// TwinCAT 3 PLC project PulsedPowerSlim_PLC
// ProgramVersion: 3.1.4023.0
// libraries:
//   Tc2_DataExchange, * (Beckhoff Automation GmbH)
//   Tc2_Math, * (Beckhoff Automation GmbH)
//   Tc2_Standard, * (Beckhoff Automation GmbH)
//   Tc2_System, * (Beckhoff Automation GmbH)
//   Tc3_EventLogger, * (Beckhoff Automation GmbH)
//   Tc3_Module, * (Beckhoff Automation GmbH)
// project tree:
//   DUTs/ E_PulseState.TcDUT, ST_Alarm_Base.TcDUT (not stored), ST_RelayFaults_Form.TcDUT, ST_Section_Base.TcDUT, ST_Charger_Base.TcDUT, ST_FieldDevices_Base.TcDUT, ST_InstrumentReading.TcDUT, ST_RelayFaults_Base.TcDUT, ST_FieldDevices_Form.TcDUT, ST_Trip_Base.TcDUT, ST_VoltageFeedback.TcDUT (not stored)
//   GVLs/ Alarms_DB.TcGVL, GVL.TcGVL, Input.TcGVL, LCP.TcGVL (not stored), MCP_IO.TcGVL, Output.TcGVL, Permissives_DB.TcGVL, Trips_DB.TcGVL
//   / PlcTask.TcTTO
//   POUs/ Alarms.TcPOU, Alarms_FB.TcPOU (not stored), Alias.TcPOU, Heartbeat.TcPOU (not stored), MAIN.TcPOU, Permissives.TcPOU, Sequence.TcPOU, Trips.TcPOU
// real-time tasks:
//   TASK PlcTask: cycle T#10ms, priority 20, ADS port 350

CONFIGURATION PulsedPowerSlim_PLC
    RESOURCE PLC ON TwinCAT3
        TASK PlcTask(INTERVAL := T#10ms, PRIORITY := 20);
        PROGRAM MAIN WITH PlcTask : MAIN;
    END_RESOURCE
END_CONFIGURATION

// ---- DUTs/E_PulseState.TcDUT
{attribute 'qualified_only'}
{attribute 'strict'}
TYPE E_PulseState :
(
	SAFE			:= 0, //IDLE
	CHARGING		:= 1, //Charge
	CHARGECOMPLETE	:= 2, //EOC
	//DISCONNECTING	:= 3, //Disconnect
	DUMPING			:= 4, 
	//ABORT			:= 5,
	TRIPPED			:= 6	
);
END_TYPE

// ---- DUTs/ST_RelayFaults_Form.TcDUT
TYPE ST_RelayFaults_Form EXTENDS ST_RelayFaults_Base :
STRUCT
	PreFormChrgRlyFailed				: BOOL;
	PreFormChrgRlyFaultDelay_TON		: TON;
	FormTrigChrgRlyFailed				: BOOL;
	FormTrigChrgRlyFaultDelay_TON		: TON;
	PreFormTrigChrgRlyFailed			: BOOL;
	PreFormTrigChrgRlyFaultDelay_TON	: TON;
	PreFormDumpRlyFailed				: BOOL;
	PreFormDumpRlyFaultDelay_TON		: TON;
	FormTrigDumpRly1Failed				: BOOL;
	FormTrigDumpRlyFaultDelay_TON		: TON;
	PreFormTrigDumpRly1Failed			: BOOL;
	PreFormTrigDumpRlyFaultDelay_TON	: TON;
END_STRUCT
END_TYPE

// ---- DUTs/ST_Section_Base.TcDUT
//Base coil type with all the Common functionality
TYPE ST_Section_Base :
STRUCT
	
	Peak : ST_FieldDevices_Base;
	Sust : ST_FieldDevices_Base;
	Form : ST_FieldDevices_Form;
	
	FormTriggerCapVoltage_raw				: INT;
	PSU1_DCOK								: BOOL := FALSE;
	//Local_EstopPB_Pressed					: BOOL;  //NC
	SystemReadyToCharge						: BOOL := FALSE;
	LossPneumaticPressure					: BOOL;
	
	//*********************************************************************************
	(*ChargeVoltageFeedback					: REAL;
	ChargeVoltageFeedback_raw				: INT;
	ChargerVoltageFeedback_norm				: REAL;
	
	CurrentFeedback							: REAL;
	CurrentFeedback_raw						: INT;
	CurrentFeedback_norm					: REAL;
	
	chargerSetpoint							: INT;  //0-100% analog PWM 24V output -> (0 - 10V)
	chargerSetpoint_norm					: REAL;
	chargerSetpoint_raw						: REAL;
	currentSetpoint							: INT;  //0-100% analog PWM 24V output -> (0.5 - 4.5V)
	currentSetpoint_norm					: REAL;
	currentSetpoint_raw						: REAL;
	//currentSetpointFromMaster: REAL;

	
	DumpRelay1_closed						: BOOL;
	DumpRelay2_closed						: BOOL;
	ChargeRelay_closed						: BOOL := FALSE;
	ChargerIsEnabled						: BOOL := FALSE; //feedback from charger
	FlybackD1_Alive							: BOOL := FALSE;
	FlybackD2_Alive							: BOOL := FALSE;
	
	DumpResistorTemperatureHigh				: BOOL; 
	GroundLoopCurrentDetected				: BOOL;
	CoilTemperatureHigh						: BOOL := FALSE;
	AC_Interlock_RlyClose					: BOOL;
	
	
	OpenDumpRelays							: BOOL := FALSE;
	closeChargeRelay						: BOOL := FALSE;
	enableOutputToCharger					: BOOL := FALSE;  //output going to charger
	CloseACInterlockRly						: BOOL := FALSE;
	SystemFaulted							: BOOL := FALSE;
	SystemCharging							: BOOL := FALSE;
	
	
	CoilEnabled								: BOOL := TRUE;
	
	NumOfCap								: INT := 4;
	
	//CoilSafetyOK							: BOOL;
	ChargerWarning							: BOOL;  //comes from UltraCaps CANBUS message
	CapVoltage								: INT;   //Comes from UlgraCaps CANBUS message
	
	ChargerVoltageFault_TON : TON;
	ChargerVoltageFault_ET : TIME;
	CurrentSensorFault_TON : TON;
	CurrentSensorFault_ET : TIME;
	BfieldSensorFault_TON : TON;
	BfieldSensorFault_ET : TIME;
	
	CAN_id: INT;
	CAN_AdsAddr: AMSADDR;
	CAN_netID: AMSNETID;
	CAN_port: WORD;
	CAN_error: USINT;
	CAN_State: UINT;
	CAN_RxErrorCounter: USINT;	
	CAN_TxErrorCounter: USINT;	
	CAN_DiagFlag: BOOL;
	
	UltacCap_CAN_error: USINT;
	UltraCap_CAN_State: UINT;
	UltraCap_CAN_RxErrorCounter: USINT;	
	UltraCap_CAN_TxErrorCounter: USINT;	
	UltraCap_CAN_DiagFlag: BOOL;
	*)
		
END_STRUCT
END_TYPE

// ---- DUTs/ST_Charger_Base.TcDUT
TYPE ST_Charger_Base :
STRUCT
	//DI
	inhibited 		: BOOL;
	EndOfCharge 	: BOOL;
	HV_isON			: BOOL;
	OverTemp		: BOOL;
	InterlockOpen	: BOOL;
	LoadFaulted		: BOOL;
	SummaryFaulted	: BOOL;
	
	//DQ
	inhibit			: BOOL;
	HV_ON			: BOOL;
	
	//AI
	voltageFeedback_raw : INT;
	currentFeedback_raw : INT;
	
	//AQ
	voltageSP		: INT;
	
END_STRUCT
END_TYPE

// ---- DUTs/ST_FieldDevices_Base.TcDUT
TYPE ST_FieldDevices_Base :
STRUCT
	cap : ARRAY [1..12] OF ST_InstrumentReading;
	
	ChargeRelay1_close		:BOOL;
	ChargeRelay2_close		:BOOL;
	
	ShortContact1_close		:BOOL;
	UnshortContact1_close 	:BOOL;
	ShortContactEngaged		:BOOL;
	
	ShortContact2_close		:BOOL;
	UnshortContact2_close 	:BOOL;
	
	DumpRelay1_close		:BOOL;
	DumpRelay2_close		:BOOL;
	
	CloseChargeRelay1		:BOOL;
	CloseChargeRelay2		:BOOL;
	OpenDumpRelay1			:BOOL;
	OpenDumpRelay2			:BOOL;
	
END_STRUCT
END_TYPE

// ---- DUTs/ST_InstrumentReading.TcDUT
TYPE ST_InstrumentReading :
STRUCT
	
	(*CH00 : REAL;
	CH01 : REAL;
	CH02 : REAL;
	CH03 : REAL;
	CH04 : REAL;
	CH05 : REAL;
	CH06 : REAL;
	CH07 : REAL;
	R2_01_CH02 : REAL;
	R2_01_CH03 : REAL;
	R2_01_CH04 : REAL;
	R2_01_CH05 : REAL;
	R2_01_CH06 : REAL;
	R2_01_CH07 : REAL;*)
	voltageFeedback_raw		: INT;
	voltageFeedback_Norm 	: REAL;
	voltageFeedback 		: REAL;
	currentFeedback_raw		: INT;
	currentFeedback_Norm 	: REAL;
	currentFeedback 		: REAL;
END_STRUCT
END_TYPE

// ---- DUTs/ST_RelayFaults_Base.TcDUT
TYPE ST_RelayFaults_Base :
STRUCT
	DumpRelay1_FailtoClose		: BOOL;
	DumpRelay1_FailtoOpen		: BOOL;
	DumpRelay1_Failed			: BOOL;
	DumpRly1FaultDelay_TON 		: TON;
	DumpRly2FaultDelay_TON 		: TON;
	
	DumpRelay2_FailtoClose		: BOOL;
	DumpRelay2_FailtoOpen		: BOOL;
	DumpRelay2_Failed			: BOOL;
	
	ChargeRelay1_FailtoClose	: BOOL;
	ChargeRelay1_FailtoOpen		: BOOL;
	ChargeRelay1_Failed			: BOOL;
	ChrgRly1FaultDelay_TON	 	: TON;
	
	ChargeRelay2_FailtoClose	: BOOL;
	ChargeRelay2_FailtoOpen		: BOOL;
	ChargeRelay2_Failed			: BOOL;
	ChrgRly2FaultDelay_TON	 	: TON;
END_STRUCT
END_TYPE

// ---- DUTs/ST_FieldDevices_Form.TcDUT
TYPE ST_FieldDevices_Form EXTENDS ST_FieldDevices_Base :
STRUCT
	PreFormChargeRly_close		: BOOL;
	FormTrigChargeRly_close		: BOOL;
	PreFormTrigChargeRly_close 	: BOOL;
	PreFormDumpRly_close		: BOOL;
	FormTrigDumpRly1_close		: BOOL;
	PreFormTrigDumpRly1_close	: BOOL;
	
	ClosePreFormChargeRly		: BOOL;
	CloseFormTrigChargeRly		: BOOL;
	ClosePreFormTrigChargeRly	: BOOL;
	OpenPreFormDumpRly			: BOOL;
	OpenFormTrigDumpRly1		: BOOL;
	OpenPreFormTrigDumpRly1		: BOOL;
	
	FormTrigShortContact_close		: BOOL;
	FormTrigUnshortContact_close	: BOOL;
	FormTrigShortContactEngaged		: BOOL;
	
	PreFormTrigShortContact_close 	: BOOL;
	PreFormTrigUnShortContact_close : BOOL;
	PreFormTrigShortContactEngaged	: BOOL;
END_STRUCT
END_TYPE

// ---- DUTs/ST_Trip_Base.TcDUT
TYPE ST_Trip_Base :
STRUCT
	ChargerVoltageReadingFaulted 		: BOOL;
	CurrentReadingFaulted 		 		: BOOL;
	
	//ACInterlockRelayFailedtoClose		: BOOL;
	//ACInterlockRelayFailedtoOpen 		: BOOL;
	//ACintLockRlyCloseFaultDelay_TON		: TON;
	//ACintLockRlyOpenFaultDelay_TON		: TON;
	
	Peak 								: ST_RelayFaults_Base;
	Sust 								: ST_RelayFaults_Base;
	Form 								: ST_RelayFaults_Form;
	
	SystemTripped						: BOOL;
	LossPneumaticPressure				: BOOL;
	LossDCPower							: BOOL;
	
	(*HVisoRelayFailedToOpen		: BOOL;
	HVRelayOpenFaultDelay_TON	: TON;
	HVisoRelayFailedToClose		: BOOL;
	HVRelayCloseFaultDelay_TON	: TON;
	*)
END_STRUCT
END_TYPE

// ---- GVLs/Alarms_DB.TcGVL
{attribute 'qualified_only'}
VAR_GLOBAL
	MCP	: ST_Alarm_Base;
	Section1 : ST_Alarm_Base;
	Section2 : ST_Alarm_Base;
	Section3 : ST_Alarm_Base;
	Section4 : ST_Alarm_Base;
	
	
	AlarmWord_11 : ST_Alarm_Base;
	AlarmWord_12 : ST_Alarm_Base;
	AlarmWord_13 : ST_Alarm_Base;
	AlarmWord_14 : ST_Alarm_Base;
	AlarmWord_15 : ST_Alarm_Base;
END_VAR

// ---- GVLs/GVL.TcGVL
{attribute 'qualified_only'}
VAR_GLOBAL
	alarm_test : BOOL;
END_VAR

// ---- GVLs/Input.TcGVL
{attribute 'qualified_only'}
VAR_GLOBAL
//***MCP************************************************************************
	//EL1008 - DI1
	R1_01_00 AT	%I*: BOOL; //Master stop PB not pressed - black pb on mcp
	R1_01_01 AT	%I*: BOOL; //case Estop circuit okay (Rly1 (120vac)
	R1_01_02 AT %I*: BOOL; //Automatic Mode Selected (NO)
	R1_01_03 AT %I*: BOOL; //MCP PSU1 DC OK
	R1_01_04 AT %I*: BOOL; //Spare
	R1_01_05 AT %I*: BOOL; //Close All Charge Relays - from labview screenroom - opto - 24V
	R1_01_06 AT %I*: BOOL; //Open All dum relays
	R1_01_07 AT %I*: BOOL; //spare

	//EL1008 - DI2
	//TDK802 1
	R1_02_00 AT	%I*: BOOL; 
	R1_02_01 AT	%I*: BOOL;
	R1_02_02 AT %I*: BOOL; 
	R1_02_03 AT %I*: BOOL; 
	R1_02_04 AT %I*: BOOL; 
	R1_02_05 AT %I*: BOOL; 
	R1_02_06 AT %I*: BOOL; 
	R1_02_07 AT %I*: BOOL; //spare
	
	//EL1008 - DI3
	//TDK802 2
	R1_03_00 AT	%I*: BOOL; 
	R1_03_01 AT	%I*: BOOL;
	R1_03_02 AT %I*: BOOL; 
	R1_03_03 AT %I*: BOOL; 
	R1_03_04 AT %I*: BOOL; 
	R1_03_05 AT %I*: BOOL; 
	R1_03_06 AT %I*: BOOL; 
	R1_03_07 AT %I*: BOOL; //spare
		
	//EL1008 - DI4
	//TDK802 3
	R1_04_00 AT	%I*: BOOL; 
	R1_04_01 AT	%I*: BOOL;
	R1_04_02 AT %I*: BOOL; 
	R1_04_03 AT %I*: BOOL; 
	R1_04_04 AT %I*: BOOL; 
	R1_04_05 AT %I*: BOOL; 
	R1_04_06 AT %I*: BOOL; 
	R1_04_07 AT %I*: BOOL; //spare
	
	//EL1008 - DI5
	//TDK802 4
	R1_05_00 AT	%I*: BOOL; 
	R1_05_01 AT	%I*: BOOL;
	R1_05_02 AT %I*: BOOL; 
	R1_05_03 AT %I*: BOOL; 
	R1_05_04 AT %I*: BOOL; 
	R1_05_05 AT %I*: BOOL; 
	R1_05_06 AT %I*: BOOL; 
	R1_05_07 AT %I*: BOOL; //spare
	
	//EL1008 - DI6
	//TDK802 5
	R1_06_00 AT	%I*: BOOL; 
	R1_06_01 AT	%I*: BOOL;
	R1_06_02 AT %I*: BOOL; 
	R1_06_03 AT %I*: BOOL; 
	R1_06_04 AT %I*: BOOL; 
	R1_06_05 AT %I*: BOOL; 
	R1_06_06 AT %I*: BOOL; 
	R1_06_07 AT %I*: BOOL; //spare
	
	//EL1008 - DI7
	//TDK802 6
	R1_07_00 AT	%I*: BOOL; 
	R1_07_01 AT	%I*: BOOL;
	R1_07_02 AT %I*: BOOL; 
	R1_07_03 AT %I*: BOOL; 
	R1_07_04 AT %I*: BOOL; 
	R1_07_05 AT %I*: BOOL; 
	R1_07_06 AT %I*: BOOL; 
	R1_07_07 AT %I*: BOOL; //spare
	
	//EL1008 - DI8
	//TDK802 7
	R1_08_00 AT	%I*: BOOL; 
	R1_08_01 AT	%I*: BOOL;
	R1_08_02 AT %I*: BOOL; 
	R1_08_03 AT %I*: BOOL; 
	R1_08_04 AT %I*: BOOL; 
	R1_08_05 AT %I*: BOOL; 
	R1_08_06 AT %I*: BOOL; 
	R1_08_07 AT %I*: BOOL; //spare
	
	//EL1008 - DI9
	//TDK802 8
	R1_09_00 AT	%I*: BOOL; 
	R1_09_01 AT	%I*: BOOL;
	R1_09_02 AT %I*: BOOL; 
	R1_09_03 AT %I*: BOOL; 
	R1_09_04 AT %I*: BOOL; 
	R1_09_05 AT %I*: BOOL; 
	R1_09_06 AT %I*: BOOL; 
	R1_09_07 AT %I*: BOOL; //spare

//RACK 2
	//EL3068 - AI1
	R2_03_00 		AT %I*: INT;
	R2_03_00_Status AT %I*: WORD;

	R2_03_01 		AT %I*: INT;
	R2_03_01_Status AT %I*: WORD;

	R2_03_02 		AT %I*: INT;
	R2_03_02_Status AT %I*: WORD;

	R2_03_03 		AT %I*: INT;
	R2_03_03_Status AT %I*: WORD;

	R2_03_04 		AT %I*: INT;
	R2_03_04_Status AT %I*: WORD;

	R2_03_05 		AT %I*: INT;
	R2_03_05_Status AT %I*: WORD;

	R2_03_06 		AT %I*: INT;
	R2_03_06_Status AT %I*: WORD;

	R2_03_07 		AT %I*: INT;
	R2_03_07_Status AT %I*: WORD;


	//EL3068 - AI2
	R2_04_00 		AT %I*: INT;
	R2_04_00_Status AT %I*: WORD;

	R2_04_01 		AT %I*: INT;
	R2_04_01_Status AT %I*: WORD;

	R2_04_02 		AT %I*: INT;
	R2_04_02_Status AT %I*: WORD;

	R2_04_03 		AT %I*: INT;
	R2_04_03_Status AT %I*: WORD;

	R2_04_04 		AT %I*: INT;
	R2_04_04_Status AT %I*: WORD;

	R2_04_05 		AT %I*: INT;
	R2_04_05_Status AT %I*: WORD;

	R2_04_06 		AT %I*: INT;
	R2_04_06_Status AT %I*: WORD;

	R2_04_07 		AT %I*: INT;
	R2_04_07_Status AT %I*: WORD;

//***LCP1***BANK1 (Rack 3)********************************************************************
//EL3068 - AI1
	R3_01_00 		AT %I*: INT;
	R3_01_00_Status AT %I*: WORD;
	
	R3_01_01		AT %I*: INT;
	R3_01_01_Status AT %I*: WORD;
	
	R3_01_02 		AT %I*: INT;
	R3_01_02_Status AT %I*: WORD;
	
	R3_01_03 		AT %I*: INT;
	R3_01_03_Status AT %I*: WORD;
	
	R3_01_04 		AT %I*: INT;
	R3_01_04_Status AT %I*: WORD;
	
	R3_01_05 		AT %I*: INT;
	R3_01_05_Status AT %I*: WORD;
	
	R3_01_06 		AT %I*: INT;
	R3_01_06_Status AT %I*: WORD;
	
	R3_01_07 		AT %I*: INT;
	R3_01_07_Status AT %I*: WORD;
	
	//EL3068 - AI2
	R3_02_00 		AT %I*: INT;
	R3_02_00_Status AT %I*: WORD;
	
	R3_02_01		AT %I*: INT;
	R3_02_01_Status AT %I*: WORD;
	
	R3_02_02 		AT %I*: INT;
	R3_02_02_Status AT %I*: WORD;
	
	R3_02_03 		AT %I*: INT;
	R3_02_03_Status AT %I*: WORD;
	
	R3_02_04 		AT %I*: INT; //SPARE
	R3_02_04_Status AT %I*: WORD;
	
	R3_02_05 		AT %I*: INT; //SPARE
	R3_02_05_Status AT %I*: WORD;
	
	R3_02_06 		AT %I*: INT; //SPARE
	R3_02_06_Status AT %I*: WORD;
	
	R3_02_07 		AT %I*: INT; //SPARE
	R3_02_07_Status AT %I*: WORD;

//EL1008 - DI1
	R3_03_00 AT %I*: BOOL;
	R3_03_01 AT %I*: BOOL;
	R3_03_02 AT %I*: BOOL;
	R3_03_03 AT %I*: BOOL;
	R3_03_04 AT %I*: BOOL;
	R3_03_05 AT %I*: BOOL;
	R3_03_06 AT %I*: BOOL;
	R3_03_07 AT %I*: BOOL;
//EL1008 - DI2	
	R3_04_00 AT %I*: BOOL;
	R3_04_01 AT %I*: BOOL;
	R3_04_02 AT %I*: BOOL;
	R3_04_03 AT %I*: BOOL;
	R3_04_04 AT %I*: BOOL;
	R3_04_05 AT %I*: BOOL; 
	R3_04_06 AT %I*: BOOL; //SPARE
	R3_04_07 AT %I*: BOOL; //SPARE

//***LCP2***BANK2 (Rack 4)********************************************************************
//EL3068 - AI1
	R4_01_00 		AT %I*: INT;
	R4_01_00_Status AT %I*: WORD;
	
	R4_01_01		AT %I*: INT;
	R4_01_01_Status AT %I*: WORD;
	
	R4_01_02 		AT %I*: INT;
	R4_01_02_Status AT %I*: WORD;
	
	R4_01_03 		AT %I*: INT;
	R4_01_03_Status AT %I*: WORD;
	
	R4_01_04 		AT %I*: INT;
	R4_01_04_Status AT %I*: WORD;
	
	R4_01_05 		AT %I*: INT;
	R4_01_05_Status AT %I*: WORD;
	
	R4_01_06 		AT %I*: INT;
	R4_01_06_Status AT %I*: WORD;
	
	R4_01_07 		AT %I*: INT;
	R4_01_07_Status AT %I*: WORD;
	
	//EL3068 - AI2
	R4_02_00 		AT %I*: INT;
	R4_02_00_Status AT %I*: WORD;
	
	R4_02_01		AT %I*: INT;
	R4_02_01_Status AT %I*: WORD;
	
	R4_02_02 		AT %I*: INT;
	R4_02_02_Status AT %I*: WORD;
	
	R4_02_03 		AT %I*: INT;
	R4_02_03_Status AT %I*: WORD;
	
	R4_02_04 		AT %I*: INT; //SPARE
	R4_02_04_Status AT %I*: WORD;
	
	R4_02_05 		AT %I*: INT; //SPARE
	R4_02_05_Status AT %I*: WORD;
	
	R4_02_06 		AT %I*: INT; //SPARE
	R4_02_06_Status AT %I*: WORD;
	
	R4_02_07 		AT %I*: INT; //SPARE
	R4_02_07_Status AT %I*: WORD;

//EL1008 - DI1
	R4_03_00 AT %I*: BOOL;
	R4_03_01 AT %I*: BOOL;
	R4_03_02 AT %I*: BOOL;
	R4_03_03 AT %I*: BOOL;
	R4_03_04 AT %I*: BOOL;
	R4_03_05 AT %I*: BOOL;
	R4_03_06 AT %I*: BOOL;
	R4_03_07 AT %I*: BOOL;
//EL1008 - DI2	
	R4_04_00 AT %I*: BOOL;
	R4_04_01 AT %I*: BOOL;
	R4_04_02 AT %I*: BOOL;
	R4_04_03 AT %I*: BOOL;
	R4_04_04 AT %I*: BOOL;
	R4_04_05 AT %I*: BOOL; 
	R4_04_06 AT %I*: BOOL; //SPARE
	R4_04_07 AT %I*: BOOL; //SPARE

//***LCP3***BANK3 (Rack 5)********************************************************************
//EL3068 - AI1
	R5_01_00 		AT %I*: INT;
	R5_01_00_Status AT %I*: WORD;
	
	R5_01_01		AT %I*: INT;
	R5_01_01_Status AT %I*: WORD;
	
	R5_01_02 		AT %I*: INT;
	R5_01_02_Status AT %I*: WORD;
	
	R5_01_03 		AT %I*: INT;
	R5_01_03_Status AT %I*: WORD;
	
	R5_01_04 		AT %I*: INT;
	R5_01_04_Status AT %I*: WORD;
	
	R5_01_05 		AT %I*: INT;
	R5_01_05_Status AT %I*: WORD;
	
	R5_01_06 		AT %I*: INT;
	R5_01_06_Status AT %I*: WORD;
	
	R5_01_07 		AT %I*: INT;
	R5_01_07_Status AT %I*: WORD;
	
	//EL3068 - AI2
	R5_02_00 		AT %I*: INT;
	R5_02_00_Status AT %I*: WORD;
	
	R5_02_01		AT %I*: INT;
	R5_02_01_Status AT %I*: WORD;
	
	R5_02_02 		AT %I*: INT;
	R5_02_02_Status AT %I*: WORD;
	
	R5_02_03 		AT %I*: INT;
	R5_02_03_Status AT %I*: WORD;
	
	R5_02_04 		AT %I*: INT; //SPARE
	R5_02_04_Status AT %I*: WORD;
	
	R5_02_05 		AT %I*: INT; //SPARE
	R5_02_05_Status AT %I*: WORD;
	
	R5_02_06 		AT %I*: INT; //SPARE
	R5_02_06_Status AT %I*: WORD;
	
	R5_02_07 		AT %I*: INT; //SPARE
	R5_02_07_Status AT %I*: WORD;

//EL1008 - DI1
	R5_03_00 AT %I*: BOOL;
	R5_03_01 AT %I*: BOOL;
	R5_03_02 AT %I*: BOOL;
	R5_03_03 AT %I*: BOOL;
	R5_03_04 AT %I*: BOOL;
	R5_03_05 AT %I*: BOOL;
	R5_03_06 AT %I*: BOOL;
	R5_03_07 AT %I*: BOOL;
//EL1008 - DI2	
	R5_04_00 AT %I*: BOOL;
	R5_04_01 AT %I*: BOOL;
	R5_04_02 AT %I*: BOOL;
	R5_04_03 AT %I*: BOOL;
	R5_04_04 AT %I*: BOOL;
	R5_04_05 AT %I*: BOOL; 
	R5_04_06 AT %I*: BOOL; //SPARE
	R5_04_07 AT %I*: BOOL; //SPARE

//***LCP4***BANK4 (Rack 6)****FORMATION****************************************************************
//EL3068 - AI1
	R6_01_00 		AT %I*: INT;
	R6_01_00_Status AT %I*: WORD;
	
	R6_01_01		AT %I*: INT;
	R6_01_01_Status AT %I*: WORD;
	
	R6_01_02 		AT %I*: INT;
	R6_01_02_Status AT %I*: WORD;
	
	R6_01_03 		AT %I*: INT;
	R6_01_03_Status AT %I*: WORD;
	
	R6_01_04 		AT %I*: INT;
	R6_01_04_Status AT %I*: WORD;
	
	R6_01_05 		AT %I*: INT;
	R6_01_05_Status AT %I*: WORD;
	
	R6_01_06 		AT %I*: INT;
	R6_01_06_Status AT %I*: WORD;
	
	R6_01_07 		AT %I*: INT;
	R6_01_07_Status AT %I*: WORD;
	
	//EL3068 - AI2
	R6_02_00 		AT %I*: INT;
	R6_02_00_Status AT %I*: WORD;
	
	R6_02_01		AT %I*: INT;
	R6_02_01_Status AT %I*: WORD;
	
	R6_02_02 		AT %I*: INT;
	R6_02_02_Status AT %I*: WORD;
	
	R6_02_03 		AT %I*: INT;
	R6_02_03_Status AT %I*: WORD;
	
	R6_02_04 		AT %I*: INT; 
	R6_02_04_Status AT %I*: WORD;
	
	R6_02_05 		AT %I*: INT; //SPARE
	R6_02_05_Status AT %I*: WORD;
	
	R6_02_06 		AT %I*: INT; //SPARE
	R6_02_06_Status AT %I*: WORD;
	
	R6_02_07 		AT %I*: INT; //SPARE
	R6_02_07_Status AT %I*: WORD;

//EL1008 - DI1
	R6_03_00 AT %I*: BOOL;
	R6_03_01 AT %I*: BOOL;
	R6_03_02 AT %I*: BOOL;
	R6_03_03 AT %I*: BOOL;
	R6_03_04 AT %I*: BOOL;
	R6_03_05 AT %I*: BOOL;
	R6_03_06 AT %I*: BOOL;
	R6_03_07 AT %I*: BOOL;
//EL1008 - DI2	
	R6_04_00 AT %I*: BOOL;
	R6_04_01 AT %I*: BOOL;
	R6_04_02 AT %I*: BOOL;
	R6_04_03 AT %I*: BOOL;
	R6_04_04 AT %I*: BOOL;
	R6_04_05 AT %I*: BOOL; 
	R6_04_06 AT %I*: BOOL; 
	R6_04_07 AT %I*: BOOL; 
//EL1008 - DI3	
	R6_05_00 AT %I*: BOOL;
	R6_05_01 AT %I*: BOOL;
	R6_05_02 AT %I*: BOOL;
	R6_05_03 AT %I*: BOOL;
	R6_05_04 AT %I*: BOOL; //spare
	R6_05_05 AT %I*: BOOL; //spare
	R6_05_06 AT %I*: BOOL; //spare
	R6_05_07 AT %I*: BOOL; //spare
//EL1008 - DI4	
	R6_06_00 AT %I*: BOOL;
	R6_06_01 AT %I*: BOOL;
	R6_06_02 AT %I*: BOOL;
	R6_06_03 AT %I*: BOOL;
	R6_06_04 AT %I*: BOOL; 
	R6_06_05 AT %I*: BOOL; 
	R6_06_06 AT %I*: BOOL; 
	R6_06_07 AT %I*: BOOL; 
//EL1008 - DI5	
	R6_07_00 AT %I*: BOOL;
	R6_07_01 AT %I*: BOOL;
	R6_07_02 AT %I*: BOOL;
	R6_07_03 AT %I*: BOOL; //spare
	R6_07_04 AT %I*: BOOL; //spare
	R6_07_05 AT %I*: BOOL; //spare
	R6_07_06 AT %I*: BOOL; //spare
	R6_07_07 AT %I*: BOOL; //spare

END_VAR

// ---- GVLs/MCP_IO.TcGVL
{attribute 'qualified_only'}
VAR_GLOBAL
	MasterStopPB_Pressed		: BOOL;
	CageEstopCircuitOK			: BOOL;
	AutoModeSelected			: BOOL;
	PSU1_DCOK					: BOOL;
	MachineGNDrlyOpen			: BOOL;
	CloseAllChargeRlyCommand	: BOOL;
	OpenAllDumpRelayCommand		: BOOL;
	Charger 					: ARRAY [1..8] OF ST_Charger_Base;
	GLS1_hvON					: BOOL;
	GLS2_hvON					: BOOL;
	GLS3_hvON					: BOOL;
	LiftMachineGND				: BOOL;
	AllChargeRelaysClose		: BOOL;
	AllDumpRelaysOpen			: BOOL;
	GLS1_voltageSP				: INT;
	GLS2_voltageSP				: INT;
	GLS3_voltageSP				: INT;
	
	AllChargerInhibited			: BOOL;
	AllChargerHVisON			: BOOL;
END_VAR

// ---- GVLs/Output.TcGVL
{attribute 'qualified_only'}
VAR_GLOBAL
	//***MCP Rack 2**************************************************
	//EL2008 - DQ1
	R2_01_00 AT %Q*: BOOL;
	R2_01_01 AT %Q*: BOOL;
	R2_01_02 AT %Q*: BOOL;
	R2_01_03 AT %Q*: BOOL;
	R2_01_04 AT %Q*: BOOL;
	R2_01_05 AT %Q*: BOOL;
	R2_01_06 AT %Q*: BOOL;
	R2_01_07 AT %Q*: BOOL;
	
	//EL2008 - DQ2
	R2_02_00 AT %Q*: BOOL;
	R2_02_01 AT %Q*: BOOL;
	R2_02_02 AT %Q*: BOOL;
	R2_02_03 AT %Q*: BOOL;
	R2_02_04 AT %Q*: BOOL;
	R2_02_05 AT %Q*: BOOL;
	R2_02_06 AT %Q*: BOOL;
	R2_02_07 AT %Q*: BOOL; 
	
	//EL4008 - AQ1
	R2_05_00 AT %Q*: INT;	//Charger 1 - Voltage Setpoint
	R2_05_00_Status AT %Q*: WORD; //need to double check
	R2_05_01 AT %Q*: INT;	//Charger 2 - Voltage Setpoint
	R2_05_01_Status AT %Q*: WORD;
	R2_05_02 AT %Q*: INT;	//Charger 3 - Voltage Setpoint
	R2_05_02_Status AT %Q*: WORD;
	R2_05_03 AT %Q*: INT;	//Charger 4 - Voltage Setpoint
	R2_05_03_Status AT %Q*: WORD;
	R2_05_04 AT %Q*: INT;	//Charger 5 - Voltage Setpoint
	R2_05_04_Status AT %Q*: WORD;
	R2_05_05 AT %Q*: INT;	//Charger 6 - Voltage Setpoint
	R2_05_05_Status AT %Q*: WORD;
	R2_05_06 AT %Q*: INT;	//Charger 7 - Voltage Setpoint
	R2_05_06_Status AT %Q*: WORD;
	R2_05_07 AT %Q*: INT;	//Charger 8 - Voltage Setpoint
	R2_05_07_Status AT %Q*: WORD;

	//EL2008 - DQ3
	R2_06_00 AT %Q*: BOOL;
	R2_06_01 AT %Q*: BOOL;
	R2_06_02 AT %Q*: BOOL;
	R2_06_03 AT %Q*: BOOL;  //Lift Machine Ground
	R2_06_04 AT %Q*: BOOL;  //All charge relays closed
	R2_06_05 AT %Q*: BOOL;  //All Dump Relays Open
	R2_06_06 AT %Q*: BOOL;  //spare
	R2_06_07 AT %Q*: BOOL;  //spare 

	//EL4008 - AQ2
	R2_07_00 AT %Q*: INT;	//GLS 1 - Voltage Setpoint
	R2_07_00_Status AT %Q*: WORD; //need to double check
	R2_07_01 AT %Q*: INT;	//GLS 2 - Voltage Setpoint
	R2_07_01_Status AT %Q*: WORD;
	R2_07_02 AT %Q*: INT;	//GLS 3 - Voltage Setpoint
	R2_07_02_Status AT %Q*: WORD;
	R2_07_03 AT %Q*: INT;	//spare
	R2_07_03_Status AT %Q*: WORD;
	R2_07_04 AT %Q*: INT;	//spare
	R2_07_04_Status AT %Q*: WORD;
	R2_07_05 AT %Q*: INT;	//spare
	R2_07_05_Status AT %Q*: WORD;
	R2_07_06 AT %Q*: INT;	//spare
	R2_07_06_Status AT %Q*: WORD;
	R2_07_07 AT %Q*: INT;	//spare
	R2_07_07_Status AT %Q*: WORD;
	
	//***LCP1***BANK1 (Rack 3)********************************************************************
	//EL2008 - DQ1
	R3_05_00 AT %Q*: BOOL;
	R3_05_01 AT %Q*: BOOL;
	R3_05_02 AT %Q*: BOOL;
	R3_05_03 AT %Q*: BOOL;
	R3_05_04 AT %Q*: BOOL;
	R3_05_05 AT %Q*: BOOL;
	R3_05_06 AT %Q*: BOOL;
	R3_05_07 AT %Q*: BOOL; 
	
	//EL2008 - DQ2
	R3_06_00 AT %Q*: BOOL; //BANK 1 SYSTEM READY TO CHARGE
	R3_06_01 AT %Q*: BOOL; //spare
	R3_06_02 AT %Q*: BOOL; //spare
	R3_06_03 AT %Q*: BOOL; //spare
	R3_06_04 AT %Q*: BOOL; //spare
	R3_06_05 AT %Q*: BOOL; //spare
	R3_06_06 AT %Q*: BOOL; //spare
	R3_06_07 AT %Q*: BOOL; //spare

	//***LCP2***BANK2 (Rack 4)********************************************************************
	//EL2008 - DQ1
	R4_05_00 AT %Q*: BOOL;
	R4_05_01 AT %Q*: BOOL;
	R4_05_02 AT %Q*: BOOL;
	R4_05_03 AT %Q*: BOOL;
	R4_05_04 AT %Q*: BOOL;
	R4_05_05 AT %Q*: BOOL;
	R4_05_06 AT %Q*: BOOL;
	R4_05_07 AT %Q*: BOOL; 
	
	//EL2008 - DQ2
	R4_06_00 AT %Q*: BOOL; //BANK 2 SYSTEM READY TO CHARGE
	R4_06_01 AT %Q*: BOOL; //spare
	R4_06_02 AT %Q*: BOOL; //spare
	R4_06_03 AT %Q*: BOOL; //spare
	R4_06_04 AT %Q*: BOOL; //spare
	R4_06_05 AT %Q*: BOOL; //spare
	R4_06_06 AT %Q*: BOOL; //spare
	R4_06_07 AT %Q*: BOOL; //spare
	
	//***LCP3***BANK3 (Rack 5)********************************************************************
	//EL2008 - DQ1
	R5_05_00 AT %Q*: BOOL;
	R5_05_01 AT %Q*: BOOL;
	R5_05_02 AT %Q*: BOOL;
	R5_05_03 AT %Q*: BOOL;
	R5_05_04 AT %Q*: BOOL;
	R5_05_05 AT %Q*: BOOL;
	R5_05_06 AT %Q*: BOOL;
	R5_05_07 AT %Q*: BOOL; 
	
	//EL2008 - DQ2
	R5_06_00 AT %Q*: BOOL; //BANK 3 SYSTEM READY TO CHARGE
	R5_06_01 AT %Q*: BOOL; //spare
	R5_06_02 AT %Q*: BOOL; //spare
	R5_06_03 AT %Q*: BOOL; //spare
	R5_06_04 AT %Q*: BOOL; //spare
	R5_06_05 AT %Q*: BOOL; //spare
	R5_06_06 AT %Q*: BOOL; //spare
	R5_06_07 AT %Q*: BOOL; //spare

	//***LCP4***BANK4 (Rack 6)*******Formation*************************************************************
	//EL2008 - DQ1
	R6_06_00 AT %Q*: BOOL;
	R6_06_01 AT %Q*: BOOL;
	R6_06_02 AT %Q*: BOOL;
	R6_06_03 AT %Q*: BOOL;
	R6_06_04 AT %Q*: BOOL;
	R6_06_05 AT %Q*: BOOL;
	R6_06_06 AT %Q*: BOOL;
	R6_06_07 AT %Q*: BOOL; 
	
	//EL2008 - DQ2
	R6_07_00 AT %Q*: BOOL; 
	R6_07_01 AT %Q*: BOOL; 
	R6_07_02 AT %Q*: BOOL; 
	R6_07_03 AT %Q*: BOOL; //spare
	R6_07_04 AT %Q*: BOOL; //spare
	R6_07_05 AT %Q*: BOOL; //spare
	R6_07_06 AT %Q*: BOOL; //spare
	R6_07_07 AT %Q*: BOOL; //spare
	
END_VAR

// ---- GVLs/Permissives_DB.TcGVL
{attribute 'qualified_only'}
VAR_GLOBAL
	AllShortContactEngaged	: BOOL;
	AllDumpRelaysOpen		: BOOL;
	AllChargeRelaysClosed	: BOOL;
	
END_VAR

// ---- GVLs/Trips_DB.TcGVL
{attribute 'qualified_only'}
VAR_GLOBAL
	Section 					: ARRAY[1..4] OF ST_Trip_Base;
	MasterStopPBPressed			: BOOL;
	CaseEStopCircuitBroken		: BOOL;
	ManualModeSelected			: BOOL;
	MCPLossDCpower				: BOOL;
	MCPsystemTripped			: BOOL;
	
	AnyEstopPressed 			: BOOL;
	AllDCpsuOK					: BOOL;
	AnyChargerOverTemp			: BOOL;
	AnyChargerLoadFault			: BOOL;
	AnyChargerInterlockOpen		: BOOL;
	AnyChargerFaulted			: BOOL; // same as summary fault
	//SystemTripped 				: BOOL;
	//InstrumentationFaulted		: BOOL;
	AnyChargeRlyFail			: BOOL;
	AnyDumpRlyFail				: BOOL;
	//AnyACInterlockFail			: BOOL;
	
	NoFaultDetected				: BOOL;
	ClearAllFaults				: BOOL;
END_VAR

// ---- POUs/MAIN.TcPOU
PROGRAM MAIN
VAR
END_VAR

Alias();
Heartbeat();
Permissives();
Trips();
Alarms();
Sequence();

END_PROGRAM

// ---- POUs/Alias.TcPOU
PROGRAM Alias
VAR
END_VAR

//R1 & R2 : MCP**  
	//DI
	MCP_IO.MasterStopPB_Pressed					:= NOT Input.R1_01_00;  //NC - Master stop PB not pressed - black pb on mcp
	MCP_IO.CageEstopCircuitOK					:= Input.R1_01_01;  //case Estop circuit okay (Rly1 (120vac)
	MCP_IO.AutoModeSelected						:= Input.R1_01_02; // 0 = manual, 1=auto
	MCP_IO.PSU1_DCOK							:= Input.R1_01_03; //psu1 dc ok
	MCP_IO.MachineGNDrlyOpen					:= Input.R1_01_04; // machine ground lifted (opto board)	
	MCP_IO.CloseAllChargeRlyCommand				:= Input.R1_01_05; // command from screen room (opto)
	MCP_IO.OpenAllDumpRelayCommand				:= Input.R1_01_06; // command from screen room (opto)
	
	MCP_IO.Charger[1].inhibited					:= Input.R1_02_00; //TDK802 1
	MCP_IO.Charger[1].EndOfCharge				:= Input.R1_02_01; //TDK802 1
	MCP_IO.Charger[1].HV_isON					:= Input.R1_02_02; //TDK802 1
	MCP_IO.Charger[1].OverTemp					:= Input.R1_02_03; //TDK802 1
	MCP_IO.Charger[1].InterlockOpen				:= Input.R1_02_04; //TDK802 1
	MCP_IO.Charger[1].LoadFaulted				:= Input.R1_02_05; //TDK802 1
	MCP_IO.Charger[1].SummaryFaulted			:= Input.R1_02_06; //TDK802 1
	
	MCP_IO.Charger[2].inhibited					:= Input.R1_03_00; //TDK802 2
	MCP_IO.Charger[2].EndOfCharge				:= Input.R1_03_01; 
	MCP_IO.Charger[2].HV_isON					:= Input.R1_03_02; 
	MCP_IO.Charger[2].OverTemp					:= Input.R1_03_03; 
	MCP_IO.Charger[2].InterlockOpen				:= Input.R1_03_04; 
	MCP_IO.Charger[2].LoadFaulted				:= Input.R1_03_05; 
	MCP_IO.Charger[2].SummaryFaulted			:= Input.R1_03_06; 
	
	MCP_IO.Charger[3].inhibited					:= Input.R1_04_00; //TDK802 3
	MCP_IO.Charger[3].EndOfCharge				:= Input.R1_04_01; 
	MCP_IO.Charger[3].HV_isON					:= Input.R1_04_02; 
	MCP_IO.Charger[3].OverTemp					:= Input.R1_04_03; 
	MCP_IO.Charger[3].InterlockOpen				:= Input.R1_04_04; 
	MCP_IO.Charger[3].LoadFaulted				:= Input.R1_04_05; 
	MCP_IO.Charger[3].SummaryFaulted			:= Input.R1_04_06; 
	
	MCP_IO.Charger[4].inhibited					:= Input.R1_05_00; //TDK802 4
	MCP_IO.Charger[4].EndOfCharge				:= Input.R1_05_01; 
	MCP_IO.Charger[4].HV_isON					:= Input.R1_05_02; 
	MCP_IO.Charger[4].OverTemp					:= Input.R1_05_03; 
	MCP_IO.Charger[4].InterlockOpen				:= Input.R1_05_04; 
	MCP_IO.Charger[4].LoadFaulted				:= Input.R1_05_05; 
	MCP_IO.Charger[4].SummaryFaulted			:= Input.R1_05_06; 

	MCP_IO.Charger[5].inhibited					:= Input.R1_06_00; //TDK802 5
	MCP_IO.Charger[5].EndOfCharge				:= Input.R1_06_01; 
	MCP_IO.Charger[5].HV_isON					:= Input.R1_06_02; 
	MCP_IO.Charger[5].OverTemp					:= Input.R1_06_03; 
	MCP_IO.Charger[5].InterlockOpen				:= Input.R1_06_04; 
	MCP_IO.Charger[5].LoadFaulted				:= Input.R1_06_05; 
	MCP_IO.Charger[5].SummaryFaulted			:= Input.R1_06_06; 

	MCP_IO.Charger[6].inhibited					:= Input.R1_07_00; //TDK802 6
	MCP_IO.Charger[6].EndOfCharge				:= Input.R1_07_01; 
	MCP_IO.Charger[6].HV_isON					:= Input.R1_07_02; 
	MCP_IO.Charger[6].OverTemp					:= Input.R1_07_03; 
	MCP_IO.Charger[6].InterlockOpen				:= Input.R1_07_04; 
	MCP_IO.Charger[6].LoadFaulted				:= Input.R1_07_05; 
	MCP_IO.Charger[6].SummaryFaulted			:= Input.R1_07_06; 

	MCP_IO.Charger[7].inhibited					:= Input.R1_08_00; //TDK802 7
	MCP_IO.Charger[7].EndOfCharge				:= Input.R1_08_01; 
	MCP_IO.Charger[7].HV_isON					:= Input.R1_08_02; 
	MCP_IO.Charger[7].OverTemp					:= Input.R1_08_03; 
	MCP_IO.Charger[7].InterlockOpen				:= Input.R1_08_04; 
	MCP_IO.Charger[7].LoadFaulted				:= Input.R1_08_05; 
	MCP_IO.Charger[7].SummaryFaulted			:= Input.R1_08_06; 

	MCP_IO.Charger[8].inhibited					:= Input.R1_09_00; //TDK802 8
	MCP_IO.Charger[8].EndOfCharge				:= Input.R1_09_01; 
	MCP_IO.Charger[8].HV_isON					:= Input.R1_09_02; 
	MCP_IO.Charger[8].OverTemp					:= Input.R1_09_03; 
	MCP_IO.Charger[8].InterlockOpen				:= Input.R1_09_04; 
	MCP_IO.Charger[8].LoadFaulted				:= Input.R1_09_05; 
	MCP_IO.Charger[8].SummaryFaulted			:= Input.R1_09_06; 

	//AI
	MCP_IO.Charger[1].voltageFeedback_raw		:= Input.R2_03_00;
	MCP_IO.Charger[1].currentFeedback_raw		:= Input.R2_03_01;
	MCP_IO.Charger[2].voltageFeedback_raw		:= Input.R2_03_02;
	MCP_IO.Charger[2].currentFeedback_raw		:= Input.R2_03_03;
	MCP_IO.Charger[3].voltageFeedback_raw		:= Input.R2_03_04;
	MCP_IO.Charger[3].currentFeedback_raw		:= Input.R2_03_05;
	MCP_IO.Charger[4].voltageFeedback_raw		:= Input.R2_03_06;
	MCP_IO.Charger[4].currentFeedback_raw		:= Input.R2_03_07;
	MCP_IO.Charger[5].voltageFeedback_raw		:= Input.R2_04_00;
	MCP_IO.Charger[5].currentFeedback_raw		:= Input.R2_04_01;
	MCP_IO.Charger[6].voltageFeedback_raw		:= Input.R2_04_02;
	MCP_IO.Charger[6].currentFeedback_raw		:= Input.R2_04_03;
	MCP_IO.Charger[7].voltageFeedback_raw		:= Input.R2_04_04;
	MCP_IO.Charger[7].currentFeedback_raw		:= Input.R2_04_05;
	MCP_IO.Charger[8].voltageFeedback_raw		:= Input.R2_04_06;
	MCP_IO.Charger[8].currentFeedback_raw		:= Input.R2_04_07;
	
	//DQ
	Output.R2_01_00	:= MCP_IO.Charger[1].inhibit;
	Output.R2_01_01	:= MCP_IO.Charger[1].HV_ON;
	Output.R2_01_02	:= MCP_IO.Charger[2].inhibit;
	Output.R2_01_03	:= MCP_IO.Charger[2].HV_ON;
	Output.R2_01_04	:= MCP_IO.Charger[3].inhibit;
	Output.R2_01_05	:= MCP_IO.Charger[3].HV_ON;
	Output.R2_01_06	:= MCP_IO.Charger[4].inhibit;
	Output.R2_01_07	:= MCP_IO.Charger[4].HV_ON;
	
	Output.R2_02_00	:= MCP_IO.Charger[5].inhibit;
	Output.R2_02_01	:= MCP_IO.Charger[5].HV_ON;
	Output.R2_02_02	:= MCP_IO.Charger[6].inhibit;
	Output.R2_02_03	:= MCP_IO.Charger[6].HV_ON;
	Output.R2_02_04	:= MCP_IO.Charger[7].inhibit;
	Output.R2_02_05	:= MCP_IO.Charger[7].HV_ON;
	Output.R2_02_06	:= MCP_IO.Charger[8].inhibit;
	Output.R2_02_07	:= MCP_IO.Charger[8].HV_ON;
	
	Output.R2_06_00	:= MCP_IO.GLS1_hvON;
	Output.R2_06_01	:= MCP_IO.GLS2_hvON;
	Output.R2_06_02	:= MCP_IO.GLS3_hvON;
	Output.R2_06_03	:= MCP_IO.LiftMachineGND;
	Output.R2_06_04	:= MCP_IO.AllChargeRelaysClose; //only for slim
	Output.R2_06_05	:= MCP_IO.AllDumpRelaysOpen;  // only for slim
	
	//AQ
	Output.R2_05_00	:= MCP_IO.Charger[1].voltageSP;
	Output.R2_05_01	:= MCP_IO.Charger[2].voltageSP;
	Output.R2_05_02	:= MCP_IO.Charger[3].voltageSP;
	Output.R2_05_03	:= MCP_IO.Charger[4].voltageSP;	
	Output.R2_05_04	:= MCP_IO.Charger[5].voltageSP;
	Output.R2_05_05	:= MCP_IO.Charger[6].voltageSP;
	Output.R2_05_06	:= MCP_IO.Charger[7].voltageSP;
	Output.R2_05_07	:= MCP_IO.Charger[8].voltageSP;					
	
	Output.R2_07_00	:= MCP_IO.GLS1_voltageSP; //Form Trigger
	Output.R2_07_01	:= MCP_IO.GLS2_voltageSP;  //Preform trigger
	Output.R2_07_02	:= MCP_IO.GLS3_voltageSP; //preform cap charger

//R3 : Bank 1 (LCP1)***********************************************
	//EL3068 - AI
	LCP.Section[1].Peak.cap[1].voltageFeedback_raw := Input.R3_01_00;
	LCP.Section[1].Peak.cap[2].voltageFeedback_raw := Input.R3_01_01;
	LCP.Section[1].Peak.cap[3].voltageFeedback_raw := Input.R3_01_02;
	LCP.Section[1].Peak.cap[4].voltageFeedback_raw := Input.R3_01_03;
	LCP.Section[1].Peak.cap[5].voltageFeedback_raw := Input.R3_01_04;
	LCP.Section[1].Peak.cap[6].voltageFeedback_raw := Input.R3_01_05;
	LCP.Section[1].Peak.cap[7].voltageFeedback_raw := Input.R3_01_06;
	LCP.Section[1].Peak.cap[8].voltageFeedback_raw := Input.R3_01_07;
	LCP.Section[1].Peak.cap[9].voltageFeedback_raw := Input.R3_02_00;
	LCP.Section[1].Peak.cap[10].voltageFeedback_raw := Input.R3_02_01;
	
	LCP.Section[1].Sust.cap[1].voltageFeedback_raw := Input.R3_02_02;
	LCP.Section[1].Sust.cap[2].voltageFeedback_raw := Input.R3_02_03;
	
	//DI
	LCP.Section[1].Peak.ChargeRelay1_close 	:= Input.R3_03_00; //RLY 1A
	LCP.Section[1].Peak.ChargeRelay2_close 	:= Input.R3_03_01; //RLY 2A
	LCP.Section[1].Peak.DumpRelay1_close 	:= Input.R3_03_02; //RLY 3A
	LCP.Section[1].Peak.DumpRelay2_close	:= Input.R3_03_03; //RLY 4A
	LCP.Section[1].Sust.ChargeRelay1_close	:= Input.R3_03_04; //RLY 5A
	LCP.Section[1].Sust.ChargeRelay2_close	:= Input.R3_03_05; //RLY 6A
	LCP.Section[1].Sust.DumpRelay1_close	:= Input.R3_03_06; //RLY 7A
	LCP.Section[1].Sust.DumpRelay2_close	:= Input.R3_03_07; //RLY 8A
	
	LCP.Section[1].Peak.ShortContact1_close 	:= Input.R3_04_00; //psw1
	LCP.Section[1].Peak.UnshortContact1_close 	:= Input.R3_04_01; //psw2
	LCP.Section[1].Peak.ShortContact2_close 	:= Input.R3_04_02; //psw3
	LCP.Section[1].Peak.UnshortContact2_close 	:= Input.R3_04_03; //psw4
	LCP.Section[1].LossPneumaticPressure 		:= Input.R3_04_04; //psw5
	LCP.Section[1].PSU1_DCOK					:= Input.R3_04_05; //psu1 contact

	//DQ
	Output.R3_05_00 := LCP.Section[1].Peak.CloseChargeRelay1; //RLY1
	Output.R3_05_01 := LCP.Section[1].Peak.CloseChargeRelay2; //RLY2
	Output.R3_05_02 := LCP.Section[1].Peak.OpenDumpRelay1; //RLY3
	Output.R3_05_03 := LCP.Section[1].Peak.OpenDumpRelay2; //RLY4
	Output.R3_05_04 := LCP.Section[1].Sust.CloseChargeRelay1; //RLY5
	Output.R3_05_05 := LCP.Section[1].Sust.CloseChargeRelay2; //RLY6
	Output.R3_05_06 := LCP.Section[1].Sust.OpenDumpRelay1; //RLY7
	Output.R3_05_07 := LCP.Section[1].Sust.OpenDumpRelay2; //RLY8
	Output.R3_06_00 := LCP.Section[1].SystemReadyToCharge; //LED1

//R4 : Bank 2 (LCP2)***********************************************
	//EL3068 - AI
	LCP.Section[2].Peak.cap[1].voltageFeedback_raw := Input.R4_01_00;
	LCP.Section[2].Peak.cap[2].voltageFeedback_raw := Input.R4_01_01;
	LCP.Section[2].Peak.cap[3].voltageFeedback_raw := Input.R4_01_02;
	LCP.Section[2].Peak.cap[4].voltageFeedback_raw := Input.R4_01_03;
	LCP.Section[2].Peak.cap[5].voltageFeedback_raw := Input.R4_01_04;
	LCP.Section[2].Peak.cap[6].voltageFeedback_raw := Input.R4_01_05;
	LCP.Section[2].Peak.cap[7].voltageFeedback_raw := Input.R4_01_06;
	LCP.Section[2].Peak.cap[8].voltageFeedback_raw := Input.R4_01_07;
	LCP.Section[2].Peak.cap[9].voltageFeedback_raw := Input.R4_02_00;
	LCP.Section[2].Peak.cap[10].voltageFeedback_raw := Input.R4_02_01;
	
	LCP.Section[2].Sust.cap[1].voltageFeedback_raw := Input.R4_02_02;
	LCP.Section[2].Sust.cap[2].voltageFeedback_raw := Input.R4_02_03;
	
	//DI
	LCP.Section[2].Peak.ChargeRelay1_close 	:= Input.R4_03_00; //RLY 1A
	LCP.Section[2].Peak.ChargeRelay2_close 	:= Input.R4_03_01; //RLY 2A
	LCP.Section[2].Peak.DumpRelay1_close 	:= Input.R4_03_02; //RLY 3A
	LCP.Section[2].Peak.DumpRelay2_close	:= Input.R4_03_03; //RLY 4A
	LCP.Section[2].Sust.ChargeRelay1_close	:= Input.R4_03_04; //RLY 5A
	LCP.Section[2].Sust.ChargeRelay2_close	:= Input.R4_03_05; //RLY 6A
	LCP.Section[2].Sust.DumpRelay1_close	:= Input.R4_03_06; //RLY 7A
	LCP.Section[2].Sust.DumpRelay2_close	:= Input.R4_03_07; //RLY 8A
	
	LCP.Section[2].Peak.ShortContact1_close 	:= Input.R4_04_00; //psw1
	LCP.Section[2].Peak.UnshortContact1_close 	:= Input.R4_04_01; //psw2
	LCP.Section[2].Peak.ShortContact2_close 	:= Input.R4_04_02; //psw3
	LCP.Section[2].Peak.UnshortContact2_close 	:= Input.R4_04_03; //psw4
	LCP.Section[2].LossPneumaticPressure 		:= Input.R4_04_04; //psw5
	LCP.Section[2].PSU1_DCOK					:= Input.R4_04_05; //psu1 contact

	//DQ
	Output.R4_05_00 := LCP.Section[2].Peak.CloseChargeRelay1; //RLY1
	Output.R4_05_01 := LCP.Section[2].Peak.CloseChargeRelay2; //RLY2
	Output.R4_05_02 := LCP.Section[2].Peak.OpenDumpRelay1; //RLY3
	Output.R4_05_03 := LCP.Section[2].Peak.OpenDumpRelay2; //RLY4
	Output.R4_05_04 := LCP.Section[2].Sust.CloseChargeRelay1; //RLY5
	Output.R4_05_05 := LCP.Section[2].Sust.CloseChargeRelay2; //RLY6
	Output.R4_05_06 := LCP.Section[2].Sust.OpenDumpRelay1; //RLY7
	Output.R4_05_07 := LCP.Section[2].Sust.OpenDumpRelay2; //RLY8
	Output.R4_06_00 := LCP.Section[2].SystemReadyToCharge; //LED1

//R5 : Bank 3 (LCP3)***********************************************
	//EL3068 - AI
	LCP.Section[3].Peak.cap[1].voltageFeedback_raw := Input.R5_01_00;
	LCP.Section[3].Peak.cap[2].voltageFeedback_raw := Input.R5_01_01;
	LCP.Section[3].Peak.cap[3].voltageFeedback_raw := Input.R5_01_02;
	LCP.Section[3].Peak.cap[4].voltageFeedback_raw := Input.R5_01_03;
	LCP.Section[3].Peak.cap[5].voltageFeedback_raw := Input.R5_01_04;
	LCP.Section[3].Peak.cap[6].voltageFeedback_raw := Input.R5_01_05;
	LCP.Section[3].Peak.cap[7].voltageFeedback_raw := Input.R5_01_06;
	LCP.Section[3].Peak.cap[8].voltageFeedback_raw := Input.R5_01_07;
	LCP.Section[3].Peak.cap[9].voltageFeedback_raw := Input.R5_02_00;
	LCP.Section[3].Peak.cap[10].voltageFeedback_raw := Input.R5_02_01;
	
	LCP.Section[3].Sust.cap[1].voltageFeedback_raw := Input.R5_02_02;
	LCP.Section[3].Sust.cap[2].voltageFeedback_raw := Input.R5_02_03;
	
	//DI
	LCP.Section[3].Peak.ChargeRelay1_close 	:= Input.R5_03_00; //RLY 1A
	LCP.Section[3].Peak.ChargeRelay2_close 	:= Input.R5_03_01; //RLY 2A
	LCP.Section[3].Peak.DumpRelay1_close 	:= Input.R5_03_02; //RLY 3A
	LCP.Section[3].Peak.DumpRelay2_close	:= Input.R5_03_03; //RLY 4A
	LCP.Section[3].Sust.ChargeRelay1_close	:= Input.R5_03_04; //RLY 5A
	LCP.Section[3].Sust.ChargeRelay2_close	:= Input.R5_03_05; //RLY 6A
	LCP.Section[3].Sust.DumpRelay1_close	:= Input.R5_03_06; //RLY 7A
	LCP.Section[3].Sust.DumpRelay2_close	:= Input.R5_03_07; //RLY 8A
	
	LCP.Section[3].Peak.ShortContact1_close 	:= Input.R5_04_00; //psw1
	LCP.Section[3].Peak.UnshortContact1_close 	:= Input.R5_04_01; //psw2
	LCP.Section[3].Peak.ShortContact2_close 	:= Input.R5_04_02; //psw3
	LCP.Section[3].Peak.UnshortContact2_close 	:= Input.R5_04_03; //psw4
	LCP.Section[3].LossPneumaticPressure 		:= Input.R5_04_04; //psw5
	LCP.Section[3].PSU1_DCOK					:= Input.R5_04_05; //psu1 contact

	//DQ
	Output.R5_05_00 := LCP.Section[3].Peak.CloseChargeRelay1; //RLY1
	Output.R5_05_01 := LCP.Section[3].Peak.CloseChargeRelay2; //RLY2
	Output.R5_05_02 := LCP.Section[3].Peak.OpenDumpRelay1; //RLY3
	Output.R5_05_03 := LCP.Section[3].Peak.OpenDumpRelay2; //RLY4
	Output.R5_05_04 := LCP.Section[3].Sust.CloseChargeRelay1; //RLY5
	Output.R5_05_05 := LCP.Section[3].Sust.CloseChargeRelay2; //RLY6
	Output.R5_05_06 := LCP.Section[3].Sust.OpenDumpRelay1; //RLY7
	Output.R5_05_07 := LCP.Section[3].Sust.OpenDumpRelay2; //RLY8
	Output.R5_06_00 := LCP.Section[3].SystemReadyToCharge; //LED1

//R6 : Bank 4 (LCP4)*****Formation******************************************
	//EL3068 - AI
	LCP.Section[4].Form.cap[1].voltageFeedback_raw := Input.R6_01_00;
	LCP.Section[4].Form.cap[2].voltageFeedback_raw := Input.R6_01_01;
	LCP.Section[4].Form.cap[3].voltageFeedback_raw := Input.R6_01_02;
	LCP.Section[4].Form.cap[4].voltageFeedback_raw := Input.R6_01_03;
	LCP.Section[4].Form.cap[5].voltageFeedback_raw := Input.R6_01_04;
	LCP.Section[4].Form.cap[6].voltageFeedback_raw := Input.R6_01_05;
	LCP.Section[4].Form.cap[7].voltageFeedback_raw := Input.R6_01_06;
	LCP.Section[4].Form.cap[8].voltageFeedback_raw := Input.R6_01_07;
	
	LCP.Section[4].Form.cap[9].voltageFeedback_raw	:= Input.R6_02_00;
	LCP.Section[4].Form.cap[10].voltageFeedback_raw := Input.R6_02_01;
	LCP.Section[4].Form.cap[11].voltageFeedback_raw := Input.R6_02_02;
	LCP.Section[4].Form.cap[12].voltageFeedback_raw := Input.R6_02_03;
	LCP.Section[4].FormTriggerCapVoltage_raw		 := Input.R6_02_04;
	
	//DI
	LCP.Section[4].Form.ChargeRelay1_close			:= Input.R6_03_00;	//RLY 1A
	LCP.Section[4].Form.ChargeRelay2_close			:= Input.R6_03_01;	//RLY 2A
	LCP.Section[4].Form.PreFormChargeRly_close		:= Input.R6_03_02;	//RLY 3A	
	LCP.Section[4].Form.FormTrigChargeRly_close		:= Input.R6_03_03;	//RLY 4A
	LCP.Section[4].Form.PreFormTrigChargeRly_close	:= Input.R6_03_04;	//RLY 5A
	LCP.Section[4].Form.DumpRelay1_close			:= Input.R6_03_05;	//RLY 6A
	LCP.Section[4].Form.DumpRelay2_close			:= Input.R6_03_06;	//RLY 7A
	LCP.Section[4].Form.PreFormDumpRly_close		:= Input.R6_03_07;	//RLY 8A
	LCP.Section[4].Form.FormTrigDumpRly1_close		:= Input.R6_04_00;	//RLY 9A
	LCP.Section[4].Form.PreFormTrigDumpRly1_close	:= Input.R6_04_01;	//RLY 10A
	
	LCP.Section[4].Form.ShortContact1_close		:= Input.R6_04_02;  //psw1
	LCP.Section[4].Form.UnshortContact1_close	:= Input.R6_04_03;  //psw2
	LCP.Section[4].Form.ShortContact2_close		:= Input.R6_04_04;  //psw3
	LCP.Section[4].Form.UnshortContact2_close	:= Input.R6_04_05;  //psw4
	LCP.Section[4].Form.FormTrigShortContact_close		:= Input.R6_04_06;  //psw5
	LCP.Section[4].Form.FormTrigUnshortContact_close	:= Input.R6_04_07;  //psw6
	LCP.Section[4].Form.PreFormTrigShortContact_close	:= Input.R6_05_00;  //psw7
	LCP.Section[4].Form.PreFormTrigUnShortContact_close	:= Input.R6_05_01;  //psw8
	LCP.Section[4].LossPneumaticPressure				:= Input.R6_05_02;  //psw9
	LCP.Section[4].PSU1_DCOK							:= Input.R6_05_03;  //psu1
	
	//DQ
	Output.R6_06_00 := LCP.Section[4].Form.CloseChargeRelay1; //rly1
	Output.R6_06_01 := LCP.Section[4].Form.CloseChargeRelay2; //rly2
	Output.R6_06_02 := LCP.Section[4].Form.ClosePreFormChargeRly; //rly3
	Output.R6_06_03 := LCP.Section[4].Form.CloseFormTrigChargeRly; //rly4
	Output.R6_06_04 := LCP.Section[4].Form.ClosePreFormTrigChargeRly; //rly5
	Output.R6_06_05 := LCP.Section[4].Form.OpenDumpRelay1; //rly6
	Output.R6_06_06 := LCP.Section[4].Form.OpenDumpRelay2; //rly7
	Output.R6_06_07 := LCP.Section[4].Form.OpenPreFormDumpRly; //rly8
	
	Output.R6_07_00 := LCP.Section[4].Form.OpenFormTrigDumpRly1; //rly9
	Output.R6_07_01 := LCP.Section[4].Form.OpenPreFormTrigDumpRly1; //rly10
	Output.R6_07_02 := LCP.Section[4].SystemReadyToCharge; //LED1
	
	//InstrumentReading.R2_01_CH00 := Input.R3_01_00;
	//InstrumentReading.R2_01_CH01 := Input.R3_01_01;
	(*
	R2_01_02 		AT %I*: INT;
	R2_01_02_Status AT %I*: WORD;
	
	R2_01_03 		AT %I*: INT;
	R2_01_03_Status AT %I*: WORD;
	
	R2_01_04 		AT %I*: INT;
	R2_01_04_Status AT %I*: WORD;
	
	R2_01_05 		AT %I*: INT;
	R2_01_05_Status AT %I*: WORD;
	
	R2_01_06 		AT %I*: INT;
	R2_01_06_Status AT %I*: WORD;
	
	R2_01_07 		AT %I*: INT;
	R2_01_07_Status AT %I*: WORD;
	*)

END_PROGRAM

// ---- POUs/Permissives.TcPOU
PROGRAM Permissives
VAR
	i : INT := 1;  //for section 1 - 3 
	j : INT := 1; //for charger 1-8
	
END_VAR

//Charger summary faults
//Trips_DB.AnySummaryFault = FALSE AND Trips_DB.AnyEstopPressed //add to no fault detected.

//section ready to charge
FOR i := 1 TO 3 BY 1 DO
	IF Trips_DB.NoFaultDetected = TRUE AND //MCP_IO.Charger[1-8].HVisOn AND
		Permissives_DB.AllChargeRelaysClosed = TRUE AND
		LCP.Section[i].Peak.ShortContactEngaged = FALSE AND
		LCP.Section[i].Sust.ShortContactEngaged = FALSE
	THEN
		LCP.Section[i].SystemReadyToCharge := TRUE;	
	ELSE
		LCP.Section[i].SystemReadyToCharge := FALSE;		
	END_IF;
END_FOR;

//Section 4
IF Trips_DB.NoFaultDetected = TRUE AND //MCP_IO.Charger[1-8].HVisOn AND
	Permissives_DB.AllChargeRelaysClosed = TRUE AND
	LCP.Section[4].Form.ShortContactEngaged = FALSE AND
	LCP.Section[4].Form.FormTrigShortContactEngaged = FALSE AND
	LCP.Section[4].Form.PreFormTrigShortContactEngaged = FALSE 
	THEN
		LCP.Section[4].SystemReadyToCharge := TRUE;
	ELSE
		LCP.Section[4].SystemReadyToCharge := FALSE;
END_IF;
	



// shorts and unshorts
//Peaking  -- short contacts are NO, so if close is false, it is and unshort is true, then it is not shorted 
FOR i := 1 TO 3 BY 1 DO
	IF LCP.Section[i].Peak.ShortContact1_close = FALSE AND LCP.Section[i].Peak.UnshortContact1_close = TRUE AND
		LCP.Section[i].Peak.ShortContact2_close = FALSE AND LCP.Section[i].Peak.UnshortContact2_close = TRUE 
		THEN
			LCP.Section[i].Peak.ShortContactEngaged := FALSE;
		ELSE
			LCP.Section[i].Peak.ShortContactEngaged := TRUE;
	END_IF;
END_FOR;

//Sustain
FOR i := 1 TO 3 BY 1 DO
	IF LCP.Section[i].Sust.ShortContact1_close = FALSE AND LCP.Section[i].Sust.UnshortContact1_close = TRUE AND
		LCP.Section[i].Sust.ShortContact2_close = FALSE AND LCP.Section[i].Sust.UnshortContact2_close = TRUE 
		THEN
			LCP.Section[i].Sust.ShortContactEngaged := FALSE;
		ELSE
			LCP.Section[i].Sust.ShortContactEngaged := TRUE;
	END_IF;
END_FOR;

//Formation
IF LCP.Section[4].Form.ShortContact1_close = FALSE AND LCP.Section[4].Form.UnshortContact1_close = TRUE AND
	LCP.Section[4].Form.ShortContact2_close = FALSE AND LCP.Section[4].Form.UnshortContact2_close = TRUE 
	THEN
		LCP.Section[4].Form.ShortContactEngaged := FALSE;
	ELSE
		LCP.Section[4].Form.ShortContactEngaged := TRUE; //might need to clarify on the NC of the short contacts.
END_IF;
// form trig short 
IF LCP.Section[4].Form.FormTrigShortContact_close = FALSE AND LCP.Section[4].Form.FormTrigUnShortContact_close = TRUE
	THEN
		LCP.Section[4].Form.FormTrigShortContactEngaged := FALSE;
	ELSE
		LCP.Section[4].Form.FormTrigShortContactEngaged := TRUE;
END_IF
// preform trig short 
IF LCP.Section[4].Form.PreFormTrigShortContact_close = FALSE AND LCP.Section[4].Form.PreFormTrigUnShortContact_close = TRUE
	THEN
		LCP.Section[4].Form.PreFormTrigShortContactEngaged := FALSE;
	ELSE
		LCP.Section[4].Form.PreFormTrigShortContactEngaged := TRUE;
END_IF

//any short contact engaged

IF LCP.Section[1].Peak.ShortContactEngaged = TRUE AND 
	LCP.Section[2].Peak.ShortContactEngaged = TRUE AND
	LCP.Section[3].Peak.ShortContactEngaged = TRUE AND
	LCP.Section[1].Sust.ShortContactEngaged = TRUE AND
	LCP.Section[2].Sust.ShortContactEngaged = TRUE AND 
	LCP.Section[3].Sust.ShortContactEngaged = TRUE AND 
	LCP.Section[4].Form.ShortContactEngaged = TRUE AND 
	LCP.Section[4].Form.FormTrigShortContactEngaged = TRUE AND //
	LCP.Section[4].Form.PreFormTrigShortContactEngaged = TRUE //
	THEN
		Permissives_DB.AllShortContactEngaged := TRUE;
	ELSE 
		Permissives_DB.AllShortContactEngaged := FALSE;	
END_IF;

//All charger inhibited
IF MCP_IO.Charger[1].inhibited = TRUE AND
	MCP_IO.Charger[2].inhibited = TRUE AND
	MCP_IO.Charger[3].inhibited = TRUE AND
	MCP_IO.Charger[4].inhibited = TRUE AND
	MCP_IO.Charger[5].inhibited = TRUE AND
	MCP_IO.Charger[6].inhibited = TRUE AND
	MCP_IO.Charger[7].inhibited = TRUE AND
	MCP_IO.Charger[8].inhibited = TRUE 
	THEN
		MCP_IO.AllChargerInhibited := TRUE;
		ELSE
			MCP_IO.AllChargerInhibited := FALSE;
END_IF;

//All charger HV ON
IF MCP_IO.Charger[1].HV_isON = TRUE AND
	MCP_IO.Charger[2].HV_isON = TRUE AND
	MCP_IO.Charger[3].HV_isON = TRUE AND
	MCP_IO.Charger[4].HV_isON = TRUE AND
	MCP_IO.Charger[5].HV_isON = TRUE AND
	MCP_IO.Charger[6].HV_isON = TRUE AND
	MCP_IO.Charger[7].HV_isON = TRUE AND
	MCP_IO.Charger[8].HV_isON = TRUE 
	THEN
		MCP_IO.AllChargerHVisON := TRUE;
		ELSE
			MCP_IO.AllChargerHVisON := FALSE;
END_IF;


//All charge relay close
IF LCP.Section[1].Peak.ChargeRelay1_close = TRUE AND
	LCP.Section[1].Peak.ChargeRelay2_close = TRUE AND
	LCP.Section[1].Sust.ChargeRelay1_close = TRUE AND
	LCP.Section[1].Sust.ChargeRelay2_close = TRUE AND
	LCP.Section[2].Peak.ChargeRelay1_close = TRUE AND
	LCP.Section[2].Peak.ChargeRelay2_close = TRUE AND
	LCP.Section[2].Sust.ChargeRelay1_close = TRUE AND
	LCP.Section[2].Sust.ChargeRelay2_close = TRUE AND
	LCP.Section[3].Peak.ChargeRelay1_close = TRUE AND
	LCP.Section[3].Peak.ChargeRelay2_close = TRUE AND
	LCP.Section[3].Sust.ChargeRelay1_close = TRUE AND
	LCP.Section[3].Sust.ChargeRelay2_close = TRUE AND
	
	LCP.Section[4].Form.ChargeRelay1_close = TRUE AND
	LCP.Section[4].Form.ChargeRelay2_close = TRUE AND						
	LCP.Section[4].Form.PreFormChargeRly_close = TRUE AND
	LCP.Section[4].Form.FormTrigChargeRly_close = TRUE AND
	LCP.Section[4].Form.PreFormTrigChargeRly_close = TRUE 
	THEN
		Permissives_DB.AllChargeRelaysClosed := TRUE;
	ELSE
		Permissives_DB.AllChargeRelaysClosed := FALSE;
END_IF;

//All Dump relays open  ******
IF LCP.Section[1].Peak.DumpRelay1_close = FALSE AND
	LCP.Section[1].Peak.DumpRelay2_close = FALSE AND
	LCP.Section[1].Sust.DumpRelay1_close = FALSE AND
	LCP.Section[1].Sust.DumpRelay2_close = FALSE AND
	LCP.Section[2].Peak.DumpRelay1_close = FALSE AND
	LCP.Section[2].Peak.DumpRelay2_close = FALSE AND
	LCP.Section[2].Sust.DumpRelay1_close = FALSE AND
	LCP.Section[2].Sust.DumpRelay2_close = FALSE AND
	LCP.Section[3].Peak.DumpRelay1_close = FALSE AND
	LCP.Section[3].Peak.DumpRelay2_close = FALSE AND
	LCP.Section[3].Sust.DumpRelay1_close = FALSE AND
	LCP.Section[3].Sust.DumpRelay2_close = FALSE AND
	
	LCP.Section[4].Form.DumpRelay1_close = FALSE AND
	LCP.Section[4].Form.DumpRelay2_close = FALSE AND						
	LCP.Section[4].Form.PreFormDumpRly_close = FALSE AND
	LCP.Section[4].Form.FormTrigDumpRly1_close = FALSE AND
	LCP.Section[4].Form.PreFormTrigDumpRly1_close = FALSE 
	THEN
		Permissives_DB.AllDumpRelaysOpen := TRUE;
	ELSE
		Permissives_DB.AllDumpRelaysOpen := FALSE;
END_IF;


IF i > 3 THEN
	i := 1;
END_IF;


IF j > 8 THEN
	j := 1;
END_IF;

END_PROGRAM

// ---- POUs/Trips.TcPOU
PROGRAM Trips
VAR
	bTest							: BOOL;
	//delay2s : Delay2s;
	evtLogger						: FB_TcEventLogger;
	
	ACintLockRlyFaultDelay_PT		: TIME := T#2S;
	DumpRlyFaultDelay_PT			: TIME := T#2S;
	//DumpRly2FaultDelay_PT			: TIME := T#2S;
	ChrgRlyFaultDelay_PT			: TIME := T#1S;
	
	i : INT := 1;  //charger 1-8
	j : INT := 1; //section 1-3
	k : INT := 1; //section 1-4, might not need 
END_VAR


//MCP Input Trips
IF MCP_IO.MasterStopPB_Pressed = TRUE THEN
	Trips_DB.MasterStopPBPressed := TRUE;	
END_IF;

IF MCP_IO.CageEstopCircuitOK = FALSE THEN
	Trips_DB.CaseEStopCircuitBroken := TRUE; 
END_IF;

IF MCP_IO.AutoModeSelected = FALSE THEN
	Trips_DB.ManualModeSelected := TRUE; //may not be a trip
	ELSE
		Trips_DB.ManualModeSelected := FALSE;
END_IF;

IF MCP_IO.PSU1_DCOK = FALSE THEN
	Trips_DB.MCPLossDCpower := TRUE; 
END_IF;

// mapping pnumatic and dc power to trips
FOR k := 1 TO 4 BY 1 DO
	Trips_DB.Section[k].LossPneumaticPressure := LCP.Section[k].LossPneumaticPressure;
	Trips_DB.Section[k].LossDCPower := NOT LCP.Section[k].PSU1_DCOK;
END_FOR;


//any charge relay fail
IF Trips_DB.Section[1].Peak.ChargeRelay1_Failed = TRUE OR
	Trips_DB.Section[1].Peak.ChargeRelay2_Failed = TRUE OR
	Trips_DB.Section[1].Sust.ChargeRelay1_Failed = TRUE OR
	Trips_DB.Section[1].Sust.ChargeRelay2_Failed = TRUE OR
	Trips_DB.Section[2].Peak.ChargeRelay1_Failed = TRUE OR
	Trips_DB.Section[2].Peak.ChargeRelay2_Failed = TRUE OR
	Trips_DB.Section[2].Sust.ChargeRelay1_Failed = TRUE OR
	Trips_DB.Section[2].Sust.ChargeRelay2_Failed = TRUE OR
	Trips_DB.Section[3].Peak.ChargeRelay1_Failed = TRUE OR
	Trips_DB.Section[3].Peak.ChargeRelay2_Failed = TRUE OR
	Trips_DB.Section[3].Sust.ChargeRelay1_Failed = TRUE OR
	Trips_DB.Section[3].Sust.ChargeRelay2_Failed = TRUE OR
	Trips_DB.Section[4].Form.ChargeRelay1_Failed = TRUE OR 
	Trips_DB.Section[4].Form.ChargeRelay2_Failed = TRUE OR 
	Trips_DB.Section[4].Form.PreFormChrgRlyFailed = TRUE OR 
	Trips_DB.Section[4].Form.FormTrigChrgRlyFailed = TRUE OR
	Trips_DB.Section[4].Form.PreFormTrigChrgRlyFailed = TRUE		
	THEN 
		Trips_DB.AnyChargeRlyFail := TRUE;
	ELSE
		Trips_DB.AnyChargeRlyFail := FALSE;
END_IF;

//any dump relay fail
IF Trips_DB.Section[1].Peak.DumpRelay1_Failed = TRUE OR
	Trips_DB.Section[1].Peak.DumpRelay2_Failed = TRUE OR
	Trips_DB.Section[1].Sust.DumpRelay1_Failed = TRUE OR
	Trips_DB.Section[1].Sust.DumpRelay2_Failed = TRUE OR
	Trips_DB.Section[2].Peak.DumpRelay1_Failed = TRUE OR
	Trips_DB.Section[2].Peak.DumpRelay2_Failed = TRUE OR
	Trips_DB.Section[2].Sust.DumpRelay1_Failed = TRUE OR
	Trips_DB.Section[2].Sust.DumpRelay2_Failed = TRUE OR
	Trips_DB.Section[3].Peak.DumpRelay1_Failed = TRUE OR
	Trips_DB.Section[3].Peak.DumpRelay2_Failed = TRUE OR
	Trips_DB.Section[3].Sust.DumpRelay1_Failed = TRUE OR
	Trips_DB.Section[3].Sust.DumpRelay2_Failed = TRUE OR
	Trips_DB.Section[4].Form.DumpRelay1_Failed = TRUE OR 
	Trips_DB.Section[4].Form.DumpRelay2_Failed = TRUE OR 
	Trips_DB.Section[4].Form.PreFormDumpRlyFailed = TRUE OR 
	Trips_DB.Section[4].Form.FormTrigDumpRly1Failed = TRUE OR
	Trips_DB.Section[4].Form.PreFormTrigDumpRly1Failed = TRUE		
	THEN 
		Trips_DB.AnyDumpRlyFail := TRUE;
	ELSE
		Trips_DB.AnyDumpRlyFail := FALSE;
END_IF;

//if relays failed, chargers faulted, loss pneumatic pressure, or loss dc power then 
//Trips_DB.Section[j].SystemTripped := TRUE;

//system trip 
//section 1-3
FOR j := 1 TO 3 BY 1 DO
	IF Trips_DB.Section[j].LossDCPower = TRUE OR 
		Trips_DB.Section[j].LossPneumaticPressure = TRUE OR
		Trips_DB.Section[j].Peak.ChargeRelay1_Failed = TRUE OR
		Trips_DB.Section[j].Peak.ChargeRelay2_Failed = TRUE OR
		Trips_DB.Section[j].Peak.DumpRelay1_Failed = TRUE OR
		Trips_DB.Section[j].Peak.DumpRelay2_Failed = TRUE OR
		Trips_DB.Section[j].Sust.ChargeRelay1_Failed = TRUE OR
		Trips_DB.Section[j].Sust.ChargeRelay2_Failed = TRUE OR
		Trips_DB.Section[j].Sust.DumpRelay1_Failed = TRUE OR
		Trips_DB.Section[j].Sust.DumpRelay2_Failed = TRUE 
		// shorted when not supposed to ?
		THEN
			Trips_DB.Section[j].SystemTripped := TRUE;
	END_IF;
END_FOR;

//formation
IF Trips_DB.Section[4].LossDCPower = TRUE OR 
	Trips_DB.Section[4].LossPneumaticPressure = TRUE OR
	Trips_DB.Section[4].Form.ChargeRelay1_Failed = TRUE OR
	Trips_DB.Section[4].Form.ChargeRelay2_Failed = TRUE OR
	Trips_DB.Section[4].Form.DumpRelay1_Failed = TRUE OR
	Trips_DB.Section[4].Form.DumpRelay2_Failed = TRUE OR
	Trips_DB.Section[4].Form.PreFormChrgRlyFailed = TRUE OR
	Trips_DB.Section[4].Form.FormTrigChrgRlyFailed = TRUE OR
	Trips_DB.Section[4].Form.PreFormTrigChrgRlyFailed = TRUE OR
	Trips_DB.Section[4].Form.PreFormDumpRlyFailed = TRUE OR
	Trips_DB.Section[4].Form.FormTrigDumpRly1Failed = TRUE OR
	Trips_DB.Section[4].Form.PreFormTrigDumpRly1Failed = TRUE
	THEN
		Trips_DB.Section[4].SystemTripped := TRUE;
END_IF;


//Charger faults
FOR i := 1 TO 8 BY 1 DO
	//OVERTEMP 
	IF MCP_IO.Charger[i].OverTemp = TRUE THEN
		Trips_DB.AnyChargerOverTemp := TRUE;  
	END_IF;
	//Load faults
	IF MCP_IO.Charger[i].LoadFaulted = TRUE THEN
		Trips_DB.AnyChargerLoadFault := TRUE;  
	END_IF;
	//Interlock Open
	IF MCP_IO.Charger[i].InterlockOpen = TRUE THEN
		Trips_DB.AnyChargerInterlockOpen := TRUE;  
	END_IF;
	
END_FOR;

//Charger summary faults
FOR i := 1 TO 8 BY 1 DO
	IF MCP_IO.Charger[i].SummaryFaulted = TRUE THEN
		Trips_DB.AnyChargerFaulted := TRUE;  
	END_IF;
END_FOR;

//MCP trip
IF Trips_DB.AnyChargerFaulted = TRUE OR 
	Trips_DB.MasterStopPBPressed = TRUE OR
	Trips_DB.CaseEStopCircuitBroken = TRUE OR
	Trips_DB.MCPLossDCpower = TRUE 
	THEN
		Trips_DB.MCPsystemTripped := TRUE;
END_IF


//*******************E-Stop Trips
IF MCP_IO.MasterStopPB_Pressed = TRUE OR MCP_IO.CageEstopCircuitOK THEN
	Trips_DB.AnyEstopPressed := TRUE;  
END_IF;	

//*********************DC PSU
IF MCP_IO.PSU1_DCOK = TRUE AND 
	LCP.Section[1].PSU1_DCOK = TRUE AND
	LCP.Section[2].PSU1_DCOK = TRUE AND
	LCP.Section[3].PSU1_DCOK = TRUE AND
	LCP.Section[4].PSU1_DCOK = TRUE 
	THEN
		TRIPS_DB.AllDCpsuOK := TRUE;
	ELSE 
		TRIPS_DB.AllDCpsuOK := FALSE;
END_IF;

//Relay faults***************************************
//section 1 - 3
FOR j := 1 TO 3 BY 1 DO
	//Peak Charge rly1
		//fail to close
	IF LCP.Section[j].Peak.CloseChargeRelay1 = TRUE AND LCP.Section[j].Peak.ChargeRelay1_close = FALSE THEN 
		//start timer
		Trips_DB.Section[j].Peak.ChrgRly1FaultDelay_TON (IN:= TRUE, PT := ChrgRlyFaultDelay_PT);
		
		IF Trips_DB.Section[j].Peak.ChrgRly1FaultDelay_TON.Q = TRUE THEN 
			Trips_DB.Section[j].Peak.ChargeRelay1_FailtoClose := TRUE; 
			Trips_DB.Section[j].Peak.ChrgRly1FaultDelay_TON (IN:= FALSE);
		END_IF;
	ELSE
		Trips_DB.Section[j].Peak.ChrgRly1FaultDelay_TON (IN:= FALSE);
	END_IF;

		//fail to open
	IF LCP.Section[j].Peak.CloseChargeRelay1 = FALSE AND LCP.Section[j].Peak.ChargeRelay1_close = TRUE THEN 
		//start timer
		Trips_DB.Section[j].Peak.ChrgRly1FaultDelay_TON (IN:= TRUE, PT := ChrgRlyFaultDelay_PT);
		
		IF Trips_DB.Section[j].Peak.ChrgRly1FaultDelay_TON.Q = TRUE THEN 
			Trips_DB.Section[j].Peak.ChargeRelay1_FailtoOpen := TRUE; 
			Trips_DB.Section[j].Peak.ChrgRly1FaultDelay_TON (IN:= FALSE);
		END_IF;
	ELSE
		Trips_DB.Section[j].Peak.ChrgRly1FaultDelay_TON (IN:= FALSE);
	
	END_IF;

	//Peak Charge rly2	
		//fail to close
	IF LCP.Section[j].Peak.CloseChargeRelay2 = TRUE AND LCP.Section[j].Peak.ChargeRelay2_close = FALSE THEN 
		//start timer
		Trips_DB.Section[j].Peak.ChrgRly2FaultDelay_TON (IN:= TRUE, PT := ChrgRlyFaultDelay_PT);
		
		IF Trips_DB.Section[j].Peak.ChrgRly2FaultDelay_TON.Q = TRUE THEN 
			Trips_DB.Section[j].Peak.ChargeRelay2_FailtoClose := TRUE; 
			Trips_DB.Section[j].Peak.ChrgRly2FaultDelay_TON (IN:= FALSE);
		END_IF;
	ELSE
		Trips_DB.Section[j].Peak.ChrgRly2FaultDelay_TON (IN:= FALSE);
	END_IF;
	
		//fail to open
	IF LCP.Section[j].Peak.CloseChargeRelay2 = FALSE AND LCP.Section[j].Peak.ChargeRelay2_close = TRUE THEN 
		//start timer
		Trips_DB.Section[j].Peak.ChrgRly2FaultDelay_TON (IN:= TRUE, PT := ChrgRlyFaultDelay_PT);
		
		IF Trips_DB.Section[j].Peak.ChrgRly2FaultDelay_TON.Q = TRUE THEN 
			Trips_DB.Section[j].Peak.ChargeRelay2_FailtoOpen := TRUE; 
			Trips_DB.Section[j].Peak.ChrgRly2FaultDelay_TON (IN:= FALSE);
		END_IF;
	ELSE
		Trips_DB.Section[j].Peak.ChrgRly2FaultDelay_TON (IN:= FALSE);
	END_IF;

	//Peak dump rly1
		//fail to open
	IF LCP.Section[j].Peak.OpenDumpRelay1 = TRUE AND LCP.Section[j].Peak.DumpRelay1_close = TRUE THEN 
		//start timer
		Trips_DB.Section[j].Peak.DumpRly1FaultDelay_TON (IN := TRUE, PT := DumpRlyFaultDelay_PT);

		IF Trips_DB.Section[j].Peak.DumpRly1FaultDelay_TON.Q = TRUE THEN 
			Trips_DB.Section[j].Peak.DumpRelay1_FailtoOpen := TRUE; 
			Trips_DB.Section[j].Peak.DumpRly1FaultDelay_TON (IN:= FALSE);
		END_IF; 
	ELSE
		Trips_DB.Section[j].Peak.DumpRly1FaultDelay_TON (IN:= FALSE);
	END_IF;

		//fail to close
	IF LCP.Section[j].Peak.OpenDumpRelay1 = FALSE AND LCP.Section[j].Peak.DumpRelay1_close = FALSE THEN 
		//start timer
		Trips_DB.Section[j].Peak.DumpRly1FaultDelay_TON (IN := TRUE, PT := DumpRlyFaultDelay_PT); 
		
		IF Trips_DB.Section[j].Peak.DumpRly1FaultDelay_TON.Q = TRUE THEN 
			Trips_DB.Section[j].Peak.DumpRelay1_FailtoClose := TRUE;
			Trips_DB.Section[j].Peak.DumpRly1FaultDelay_TON (IN:= FALSE);
		END_IF;
	ELSE
		Trips_DB.Section[j].Peak.DumpRly1FaultDelay_TON (IN:= FALSE);
	END_IF;

	//Peak dump rly2
		//fail to open
	IF LCP.Section[j].Peak.OpenDumpRelay2 = TRUE AND LCP.Section[j].Peak.DumpRelay2_close = TRUE THEN 
		//start timer
		Trips_DB.Section[j].Peak.DumpRly2FaultDelay_TON (IN := TRUE, PT := DumpRlyFaultDelay_PT); 
		
		IF Trips_DB.Section[j].Peak.DumpRly2FaultDelay_TON.Q = TRUE THEN 
			Trips_DB.Section[j].Peak.DumpRelay2_FailtoOpen := TRUE; 
			Trips_DB.Section[j].Peak.DumpRly2FaultDelay_TON (IN:= FALSE);
		END_IF;
	ELSE
		Trips_DB.Section[j].Peak.DumpRly2FaultDelay_TON (IN:= FALSE);
	END_IF;

		//fail to close
	IF LCP.Section[j].Peak.OpenDumpRelay2 = FALSE AND LCP.Section[j].Peak.DumpRelay2_close = FALSE THEN 
		//start timer
		Trips_DB.Section[j].Peak.DumpRly2FaultDelay_TON (IN := TRUE, PT := DumpRlyFaultDelay_PT); 
		IF Trips_DB.Section[j].Peak.DumpRly2FaultDelay_TON.Q = TRUE THEN 
			Trips_DB.Section[j].Peak.DumpRelay2_FailtoClose := TRUE; 
			
		END_IF;
	ELSE
		Trips_DB.Section[j].Peak.DumpRly2FaultDelay_TON (IN:= FALSE);
	END_IF;
//*************************************************************************************************

//Sust Charge rly1
		//fail to close
	IF LCP.Section[j].Sust.CloseChargeRelay1 = TRUE AND LCP.Section[j].Sust.ChargeRelay1_close = FALSE THEN 
		//start timer
		Trips_DB.Section[j].Sust.ChrgRly1FaultDelay_TON (IN:= TRUE, PT := ChrgRlyFaultDelay_PT);
		
		IF Trips_DB.Section[j].Sust.ChrgRly1FaultDelay_TON.Q = TRUE THEN 
			Trips_DB.Section[j].Sust.ChargeRelay1_FailtoClose := TRUE; 
			Trips_DB.Section[j].Sust.ChrgRly1FaultDelay_TON (IN:= FALSE);
		END_IF;
	ELSE
		Trips_DB.Section[j].Sust.ChrgRly1FaultDelay_TON (IN:= FALSE);	
	END_IF;

		//fail to open
	IF LCP.Section[j].Sust.CloseChargeRelay1 = FALSE AND LCP.Section[j].Sust.ChargeRelay1_close = TRUE THEN 
		//start timer
		Trips_DB.Section[j].Sust.ChrgRly1FaultDelay_TON (IN:= TRUE, PT := ChrgRlyFaultDelay_PT);
		
		IF Trips_DB.Section[j].Sust.ChrgRly1FaultDelay_TON.Q = TRUE THEN 
			Trips_DB.Section[j].Sust.ChargeRelay1_FailtoOpen := TRUE; 
			Trips_DB.Section[j].Sust.ChrgRly1FaultDelay_TON (IN:= FALSE);
		END_IF;
	ELSE
		Trips_DB.Section[j].Sust.ChrgRly1FaultDelay_TON (IN:= FALSE);
	END_IF;

	//Sust Charge rly2	
		//fail to close
	IF LCP.Section[j].Sust.CloseChargeRelay2 = TRUE AND LCP.Section[j].Sust.ChargeRelay2_close = FALSE THEN 
		//start timer
		Trips_DB.Section[j].Sust.ChrgRly2FaultDelay_TON (IN:= TRUE, PT := ChrgRlyFaultDelay_PT);
		
		IF Trips_DB.Section[j].Sust.ChrgRly2FaultDelay_TON.Q = TRUE THEN 
			Trips_DB.Section[j].Sust.ChargeRelay2_FailtoClose := TRUE;
			Trips_DB.Section[j].Sust.ChrgRly2FaultDelay_TON (IN:= FALSE);
		END_IF;
	ELSE
		Trips_DB.Section[j].Sust.ChrgRly2FaultDelay_TON (IN:= FALSE);
	END_IF;
	
		//fail to open
	IF LCP.Section[j].Sust.CloseChargeRelay2 = FALSE AND LCP.Section[j].Sust.ChargeRelay2_close = TRUE THEN 
		//start timer
		Trips_DB.Section[j].Sust.ChrgRly2FaultDelay_TON (IN:= TRUE, PT := ChrgRlyFaultDelay_PT);
		
		IF Trips_DB.Section[j].Sust.ChrgRly2FaultDelay_TON.Q = TRUE THEN 
			Trips_DB.Section[j].Sust.ChargeRelay2_FailtoOpen := TRUE; 
			Trips_DB.Section[j].Sust.ChrgRly2FaultDelay_TON (IN:= FALSE);
		END_IF;
	ELSE
		Trips_DB.Section[j].Sust.ChrgRly2FaultDelay_TON (IN:= FALSE);
	END_IF;

	//Sust dump rly1
		//fail to open
	IF LCP.Section[j].Sust.OpenDumpRelay1 = TRUE AND LCP.Section[j].Sust.DumpRelay1_close = TRUE THEN 
		//start timer
		Trips_DB.Section[j].Sust.DumpRly1FaultDelay_TON (IN := TRUE, PT := DumpRlyFaultDelay_PT);

		IF Trips_DB.Section[j].Sust.DumpRly1FaultDelay_TON.Q = TRUE THEN 
			Trips_DB.Section[j].Sust.DumpRelay1_FailtoOpen := TRUE; 
			Trips_DB.Section[j].Sust.DumpRly1FaultDelay_TON (IN:= FALSE);
		END_IF; 
	ELSE
		Trips_DB.Section[j].Sust.DumpRly1FaultDelay_TON (IN:= FALSE);
	END_IF;

		//fail to close
	IF LCP.Section[j].Sust.OpenDumpRelay1 = FALSE AND LCP.Section[j].Sust.DumpRelay1_close = FALSE THEN 
		//start timer
		Trips_DB.Section[j].Sust.DumpRly1FaultDelay_TON (IN := TRUE, PT := DumpRlyFaultDelay_PT); 
		
		IF Trips_DB.Section[j].Sust.DumpRly1FaultDelay_TON.Q = TRUE THEN 
			Trips_DB.Section[j].Sust.DumpRelay1_FailtoClose := TRUE; 
			Trips_DB.Section[j].Sust.DumpRly1FaultDelay_TON (IN:= FALSE);
		END_IF;
	ELSE
		Trips_DB.Section[j].Sust.DumpRly1FaultDelay_TON (IN:= FALSE);
	END_IF;

	//Sust dump rly2
		//fail to open
	IF LCP.Section[j].Sust.OpenDumpRelay2 = TRUE AND LCP.Section[j].Sust.DumpRelay2_close = TRUE THEN 
		//start timer
		Trips_DB.Section[j].Sust.DumpRly2FaultDelay_TON (IN := TRUE, PT := DumpRlyFaultDelay_PT); 
		
		IF Trips_DB.Section[j].Sust.DumpRly2FaultDelay_TON.Q = TRUE THEN 
			Trips_DB.Section[j].Sust.DumpRelay2_FailtoOpen := TRUE; 
			Trips_DB.Section[j].Sust.DumpRly2FaultDelay_TON (IN:= FALSE);
		END_IF;
	ELSE
		Trips_DB.Section[j].Sust.DumpRly2FaultDelay_TON (IN:= FALSE);
	END_IF;

		//fail to close
	IF LCP.Section[j].Sust.OpenDumpRelay2 = FALSE AND LCP.Section[j].Sust.DumpRelay2_close = FALSE THEN 
		//start timer
		Trips_DB.Section[j].Sust.DumpRly2FaultDelay_TON (IN := TRUE, PT := DumpRlyFaultDelay_PT); 
		IF Trips_DB.Section[j].Sust.DumpRly2FaultDelay_TON.Q = TRUE THEN 
			Trips_DB.Section[j].Sust.DumpRelay2_FailtoClose := TRUE; 
			Trips_DB.Section[j].Sust.DumpRly2FaultDelay_TON (IN:= FALSE);
		END_IF;
	ELSE
		Trips_DB.Section[j].Sust.DumpRly2FaultDelay_TON (IN:= FALSE);
	END_IF;
	
END_FOR;
//****************************************	
	
//Form Charge rly1
		//fail to close
IF LCP.Section[4].Form.CloseChargeRelay1 = TRUE AND LCP.Section[4].Form.ChargeRelay1_close = FALSE THEN 
		//start timer
		Trips_DB.Section[4].Form.ChrgRly1FaultDelay_TON (IN:= TRUE, PT := ChrgRlyFaultDelay_PT);
		
		IF Trips_DB.Section[4].Form.ChrgRly1FaultDelay_TON.Q = TRUE THEN 
			Trips_DB.Section[4].Form.ChargeRelay1_FailtoClose := TRUE; 
			Trips_DB.Section[4].Form.ChrgRly1FaultDelay_TON (IN:= FALSE);
		END_IF;
	ELSE
		Trips_DB.Section[4].Form.ChrgRly1FaultDelay_TON (IN:= FALSE);		
END_IF;

		//fail to open
IF LCP.Section[4].Form.CloseChargeRelay1 = FALSE AND LCP.Section[4].Form.ChargeRelay1_close = TRUE THEN 
		//start timer
		Trips_DB.Section[4].Form.ChrgRly1FaultDelay_TON (IN:= TRUE, PT := ChrgRlyFaultDelay_PT);
		
		IF Trips_DB.Section[4].Form.ChrgRly1FaultDelay_TON.Q = TRUE THEN 
			Trips_DB.Section[4].Form.ChargeRelay1_FailtoOpen := TRUE; 
			Trips_DB.Section[4].Form.ChrgRly1FaultDelay_TON (IN:= FALSE);
		END_IF;
	ELSE
		Trips_DB.Section[4].Form.ChrgRly1FaultDelay_TON (IN:= FALSE);
END_IF;

	//Form Charge rly2	
		//fail to close
IF LCP.Section[4].Form.CloseChargeRelay2 = TRUE AND LCP.Section[4].Form.ChargeRelay2_close = FALSE THEN 
		//start timer
		Trips_DB.Section[4].Form.ChrgRly2FaultDelay_TON (IN:= TRUE, PT := ChrgRlyFaultDelay_PT);
		
		IF Trips_DB.Section[4].Form.ChrgRly2FaultDelay_TON.Q = TRUE THEN 
			Trips_DB.Section[4].Form.ChargeRelay2_FailtoClose := TRUE; 
			Trips_DB.Section[4].Form.ChrgRly2FaultDelay_TON (IN:= FALSE);
		END_IF;
	ELSE
		Trips_DB.Section[4].Form.ChrgRly2FaultDelay_TON (IN:= FALSE);
END_IF;
	
		//fail to open
IF LCP.Section[4].Form.CloseChargeRelay2 = FALSE AND LCP.Section[4].Form.ChargeRelay2_close = TRUE THEN 
		//start timer
		Trips_DB.Section[4].Form.ChrgRly2FaultDelay_TON (IN:= TRUE, PT := ChrgRlyFaultDelay_PT);
		
		IF Trips_DB.Section[4].Form.ChrgRly2FaultDelay_TON.Q = TRUE THEN 
			Trips_DB.Section[4].Form.ChargeRelay2_FailtoOpen := TRUE; 
			Trips_DB.Section[4].Form.ChrgRly2FaultDelay_TON (IN:= FALSE);
		END_IF;
	ELSE
		Trips_DB.Section[4].Form.ChrgRly2FaultDelay_TON (IN:= FALSE);
END_IF;

	//Form dump rly1
		//fail to open
IF LCP.Section[4].Form.OpenDumpRelay1 = TRUE AND LCP.Section[4].Form.DumpRelay1_close = TRUE THEN 
		//start timer
		Trips_DB.Section[4].Form.DumpRly1FaultDelay_TON (IN := TRUE, PT := DumpRlyFaultDelay_PT);

		IF Trips_DB.Section[4].Form.DumpRly1FaultDelay_TON.Q = TRUE THEN 
			Trips_DB.Section[4].Form.DumpRelay1_FailtoOpen := TRUE; 
			Trips_DB.Section[4].Form.DumpRly1FaultDelay_TON (IN:= FALSE);
		END_IF; 
	ELSE
		Trips_DB.Section[4].Form.DumpRly1FaultDelay_TON (IN:= FALSE);
END_IF;

		//fail to close
IF LCP.Section[4].Form.OpenDumpRelay1 = FALSE AND LCP.Section[4].Form.DumpRelay1_close = FALSE THEN 
		//start timer
		Trips_DB.Section[4].Form.DumpRly1FaultDelay_TON (IN := TRUE, PT := DumpRlyFaultDelay_PT); 
		
		IF Trips_DB.Section[4].Form.DumpRly1FaultDelay_TON.Q = TRUE THEN 
			Trips_DB.Section[4].Form.DumpRelay1_FailtoClose := TRUE; 
			Trips_DB.Section[4].Form.DumpRly1FaultDelay_TON (IN:= FALSE);
		END_IF;
	ELSE
		Trips_DB.Section[4].Form.DumpRly1FaultDelay_TON (IN:= FALSE);
END_IF;

	//Form dump rly2
		//fail to open
IF LCP.Section[4].Form.OpenDumpRelay2 = TRUE AND LCP.Section[4].Form.DumpRelay2_close = TRUE THEN 
		//start timer
		Trips_DB.Section[4].Form.DumpRly2FaultDelay_TON (IN := TRUE, PT := DumpRlyFaultDelay_PT); 
		
		IF Trips_DB.Section[4].Form.DumpRly2FaultDelay_TON.Q = TRUE THEN 
			Trips_DB.Section[4].Form.DumpRelay2_FailtoOpen := TRUE; 
			Trips_DB.Section[4].Form.DumpRly2FaultDelay_TON (IN:= FALSE);
		END_IF;
	ELSE
		Trips_DB.Section[4].Form.DumpRly2FaultDelay_TON (IN:= FALSE);
END_IF;

		//fail to close
IF LCP.Section[4].Form.OpenDumpRelay2 = FALSE AND LCP.Section[4].Form.DumpRelay2_close = FALSE THEN 
		//start timer
		Trips_DB.Section[4].Form.DumpRly2FaultDelay_TON (IN := TRUE, PT := DumpRlyFaultDelay_PT); 
		IF Trips_DB.Section[4].Form.DumpRly2FaultDelay_TON.Q = TRUE THEN 
			Trips_DB.Section[4].Form.DumpRelay2_FailtoClose := TRUE; 
			Trips_DB.Section[4].Form.DumpRly2FaultDelay_TON (IN:= FALSE);
		END_IF;
	ELSE
		Trips_DB.Section[4].Form.DumpRly2FaultDelay_TON (IN:= FALSE);
END_IF;	

	//PreForm Charge rly
		//fail to close
IF (LCP.Section[4].Form.ClosePreFormChargeRly = TRUE AND LCP.Section[4].Form.PreFormChargeRly_close = FALSE) OR 
		(LCP.Section[4].Form.ClosePreFormChargeRly = FALSE AND LCP.Section[4].Form.PreFormChargeRly_close = TRUE) 
		THEN 
		//start timer
		Trips_DB.Section[4].Form.PreFormChrgRlyFaultDelay_TON (IN:= TRUE, PT := ChrgRlyFaultDelay_PT);
		
		IF Trips_DB.Section[4].Form.PreFormChrgRlyFaultDelay_TON.Q = TRUE THEN 
			Trips_DB.Section[4].Form.PreFormChrgRlyFailed := TRUE; 
			Trips_DB.Section[4].Form.PreFormChrgRlyFaultDelay_TON (IN:= FALSE);
		END_IF;
	ELSE
		Trips_DB.Section[4].Form.PreFormChrgRlyFaultDelay_TON (IN:= FALSE);
END_IF;

//form trigger charge 
		//fail to close
IF (LCP.Section[4].Form.CloseFormTrigChargeRly = TRUE AND LCP.Section[4].Form.FormTrigChargeRly_close = FALSE) OR 
		(LCP.Section[4].Form.CloseFormTrigChargeRly = FALSE AND LCP.Section[4].Form.FormTrigChargeRly_close = TRUE) 
		THEN 
		//start timer
		Trips_DB.Section[4].Form.FormTrigChrgRlyFaultDelay_TON (IN:= TRUE, PT := ChrgRlyFaultDelay_PT);
		
		IF Trips_DB.Section[4].Form.FormTrigChrgRlyFaultDelay_TON.Q = TRUE THEN 
			Trips_DB.Section[4].Form.FormTrigChrgRlyFailed := TRUE; 
			Trips_DB.Section[4].Form.FormTrigChrgRlyFaultDelay_TON (IN:= FALSE);
		END_IF;
	ELSE
		Trips_DB.Section[4].Form.FormTrigChrgRlyFaultDelay_TON (IN:= FALSE);
END_IF;

//preform trigger charge
		//fail to close
IF (LCP.Section[4].Form.ClosePreFormTrigChargeRly = TRUE AND LCP.Section[4].Form.PreFormTrigChargeRly_close = FALSE) OR 
		(LCP.Section[4].Form.ClosePreFormTrigChargeRly = FALSE AND LCP.Section[4].Form.PreFormTrigChargeRly_close = TRUE) 
		THEN 
		//start timer
		Trips_DB.Section[4].Form.PreFormTrigChrgRlyFaultDelay_TON (IN:= TRUE, PT := ChrgRlyFaultDelay_PT);
		
		IF Trips_DB.Section[4].Form.PreFormTrigChrgRlyFaultDelay_TON.Q = TRUE THEN 
			Trips_DB.Section[4].Form.PreFormTrigChrgRlyFailed := TRUE; 
			Trips_DB.Section[4].Form.PreFormTrigChrgRlyFaultDelay_TON (IN:= FALSE);
		END_IF;
	ELSE
		Trips_DB.Section[4].Form.PreFormTrigChrgRlyFaultDelay_TON (IN:= FALSE);
END_IF;

//preform dump
	//fail to close
IF (LCP.Section[4].Form.OpenPreFormDumpRly = TRUE AND LCP.Section[4].Form.PreFormDumpRly_close = FALSE) OR 
		(LCP.Section[4].Form.OpenPreFormDumpRly = FALSE AND LCP.Section[4].Form.PreFormDumpRly_close = TRUE) 
		THEN 
		//start timer
		Trips_DB.Section[4].Form.PreFormDumpRlyFaultDelay_TON (IN:= TRUE, PT := DumpRlyFaultDelay_PT);
		
		IF Trips_DB.Section[4].Form.PreFormDumpRlyFaultDelay_TON.Q = TRUE THEN 
			Trips_DB.Section[4].Form.PreFormDumpRlyFailed := TRUE; 
			Trips_DB.Section[4].Form.PreFormDumpRlyFaultDelay_TON (IN:= FALSE);
		END_IF;
	ELSE
		Trips_DB.Section[4].Form.PreFormDumpRlyFaultDelay_TON (IN:= FALSE);
END_IF;

//form trigger dump
	//fail to close
IF (LCP.Section[4].Form.OpenFormTrigDumpRly1 = TRUE AND LCP.Section[4].Form.FormTrigDumpRly1_close = FALSE) OR 
		(LCP.Section[4].Form.OpenFormTrigDumpRly1 = FALSE AND LCP.Section[4].Form.FormTrigDumpRly1_close = TRUE) 
		THEN 
		//start timer
		Trips_DB.Section[4].Form.FormTrigDumpRlyFaultDelay_TON (IN:= TRUE, PT := DumpRlyFaultDelay_PT);
		
		IF Trips_DB.Section[4].Form.FormTrigDumpRlyFaultDelay_TON.Q = TRUE THEN 
			Trips_DB.Section[4].Form.FormTrigDumpRly1Failed := TRUE; 
			Trips_DB.Section[4].Form.FormTrigDumpRlyFaultDelay_TON (IN:= FALSE);
		END_IF;
	ELSE
		Trips_DB.Section[4].Form.FormTrigDumpRlyFaultDelay_TON (IN:= FALSE);
END_IF;
	
//preform trigger dump
	//fail to close
IF (LCP.Section[4].Form.OpenPreFormTrigDumpRly1 = TRUE AND LCP.Section[4].Form.PreFormTrigDumpRly1_close = FALSE) OR 
		(LCP.Section[4].Form.OpenPreFormTrigDumpRly1 = FALSE AND LCP.Section[4].Form.PreFormTrigDumpRly1_close = TRUE) 
		THEN 
		//start timer
		Trips_DB.Section[4].Form.PreFormTrigDumpRlyFaultDelay_TON (IN:= TRUE, PT := DumpRlyFaultDelay_PT);
		
		IF Trips_DB.Section[4].Form.PreFormTrigDumpRlyFaultDelay_TON.Q = TRUE THEN 
			Trips_DB.Section[4].Form.PreFormTrigDumpRly1Failed := TRUE; 
			Trips_DB.Section[4].Form.PreFormTrigDumpRlyFaultDelay_TON (IN:= FALSE);
		END_IF;
	ELSE
		Trips_DB.Section[4].Form.PreFormTrigDumpRlyFaultDelay_TON (IN:= FALSE);
END_IF;
	

// if rly fail to close or fail to open then trips_db.rly_failed - for alarms	
FOR j := 1 TO 3 BY 1 DO
	//peak
	IF Trips_DB.Section[j].Peak.ChargeRelay1_FailtoClose = TRUE OR Trips_DB.Section[j].Peak.ChargeRelay1_FailtoOpen = TRUE THEN
		Trips_DB.Section[j].Peak.ChargeRelay1_Failed := TRUE;  
	END_IF;
	
	IF Trips_DB.Section[j].Peak.ChargeRelay2_FailtoClose = TRUE OR Trips_DB.Section[j].Peak.ChargeRelay2_FailtoOpen = TRUE THEN
		Trips_DB.Section[j].Peak.ChargeRelay2_Failed := TRUE;  
	END_IF;
	
	IF Trips_DB.Section[j].Peak.DumpRelay1_FailtoClose = TRUE OR Trips_DB.Section[j].Peak.DumpRelay1_FailtoOpen = TRUE THEN
		Trips_DB.Section[j].Peak.DumpRelay1_Failed := TRUE;  
	END_IF;
	
	IF Trips_DB.Section[j].Peak.DumpRelay2_FailtoClose = TRUE OR Trips_DB.Section[j].Peak.DumpRelay2_FailtoOpen = TRUE THEN
		Trips_DB.Section[j].Peak.DumpRelay2_Failed := TRUE;  
	END_IF;
	
	//sust
	IF Trips_DB.Section[j].Sust.ChargeRelay1_FailtoClose = TRUE OR Trips_DB.Section[j].Sust.ChargeRelay1_FailtoOpen = TRUE THEN
		Trips_DB.Section[j].Sust.ChargeRelay1_Failed := TRUE;  
	END_IF;
	
	IF Trips_DB.Section[j].Sust.ChargeRelay2_FailtoClose = TRUE OR Trips_DB.Section[j].Sust.ChargeRelay2_FailtoOpen = TRUE THEN
		Trips_DB.Section[j].Sust.ChargeRelay2_Failed := TRUE;  
	END_IF;
	
	IF Trips_DB.Section[j].Sust.DumpRelay1_FailtoClose = TRUE OR Trips_DB.Section[j].Sust.DumpRelay1_FailtoOpen = TRUE THEN
		Trips_DB.Section[j].Sust.DumpRelay1_Failed := TRUE;  
	END_IF;
	
	IF Trips_DB.Section[j].Sust.DumpRelay2_FailtoClose = TRUE OR Trips_DB.Section[j].Sust.DumpRelay2_FailtoOpen = TRUE THEN
		Trips_DB.Section[j].Sust.DumpRelay2_Failed := TRUE;  
	END_IF;
	
END_FOR;

// no faulted detected
IF Trips_DB.MCPsystemTripped = FALSE AND
	Trips_DB.AnyChargerOverTemp = FALSE AND
	Trips_DB.AnyChargerLoadFault = FALSE AND
	Trips_DB.AnyChargerInterlockOpen = FALSE AND
	Trips_DB.AnyChargerFaulted = FALSE AND
	Trips_DB.AnyEstopPressed = FALSE AND
	Trips_DB.AnyDumpRlyFail = FALSE AND
	Trips_DB.AnyChargeRlyFail = FALSE
	THEN
		Trips_DB.NoFaultDetected := TRUE;
	ELSE
		Trips_DB.NoFaultDetected := FALSE;
END_IF;


(*
FOR i := 1 TO 10 BY 1 DO
	IF (Trips_DB.Coil[i].ACInterlockRelayFailedtoClose = TRUE OR 
		Trips_DB.Coil[i].ACInterlockRelayFailedtoOpen = TRUE OR 
		Trips_DB.Coil[i].ChargeRelay_FailtoClose = TRUE OR
		Trips_DB.Coil[i].ChargeRelay_FailtoOpen = TRUE OR
		Trips_DB.Coil[i].DumpRelay1_FailtoClose =  TRUE OR 
		Trips_DB.Coil[i].DumpRelay1_FailtoOpen = TRUE OR 
		Trips_DB.Coil[i].DumpRelay2_FailtoClose =  TRUE OR 
		Trips_DB.Coil[i].DumpRelay2_FailtoOpen = TRUE OR 
		Trips_DB.Coil[i].ChargerVoltageReadingFaulted = TRUE OR
		Trips_DB.Coil[i].CurrentReadingFaulted = TRUE OR
		Devices.Coil[i].Local_EstopPB_Pressed = TRUE OR
		Devices.Coil[i].LossPneumaticPressure = FALSE) AND Devices.Coil[i].CoilEnabled = TRUE 	
		THEN
			Devices.Coil[i].SystemFaulted := TRUE;
	END_IF
	
	IF Devices.Coil[i].SystemFaulted = TRUE THEN
		Trips_DB.SystemTripped := TRUE;
	END_IF;
END_FOR;

//*********************************** Test
(*IF InstrumentReading.R2_01_CH01 <= 0.0 THEN
	delay2s(input := FALSE);
ELSE 
	delay2s (input := TRUE);
END_IF;
bTest := delay2s.output;
*)
// Instrumentation Hardware trip
//Input.R2_01_00_Status.0;
*)
//************** Clear System Fault
IF Trips_DB.ClearAllFaults THEN
	//Trips_DB.InstrumentationFaulted := FALSE;
	//Trips_DB.SystemTripped := FALSE;
	Trips_DB.MCPsystemTripped := FALSE; //reset mcp trip
	Trips_DB.AnyChargerOverTemp := FALSE;
	Trips_DB.AnyChargerLoadFault := FALSE;  
	Trips_DB.AnyChargerInterlockOpen := FALSE;
	Trips_DB.AnyChargerFaulted := FALSE;
	Trips_DB.AnyEstopPressed := FALSE;
	Trips_DB.AnyDumpRlyFail := FALSE;
	Trips_DB.AnyChargeRlyFail := FALSE;
	Trips_DB.MasterStopPBPressed := FALSE; //this is only for alarms
	Trips_DB.CaseEStopCircuitBroken := FALSE;
	Trips_DB.MCPLossDCpower := FALSE;
	//Trips_DB.AnyACInterlockFail := FALSE;
	//reset relay trips
	FOR j := 1 TO 3 BY 1 DO 
		//reset relay faults
		Trips_DB.Section[j].SystemTripped := FALSE;
		//Peaking
		Trips_DB.Section[j].Peak.DumpRelay1_FailtoClose := FALSE;
		Trips_DB.Section[j].Peak.DumpRelay1_FailtoOpen := FALSE;
		Trips_DB.Section[j].Peak.DumpRelay2_FailtoClose := FALSE;
		Trips_DB.Section[j].Peak.DumpRelay2_FailtoOpen := FALSE;
		Trips_DB.Section[j].Peak.ChargeRelay1_FailtoClose := FALSE;
		Trips_DB.Section[j].Peak.ChargeRelay1_FailtoOpen := FALSE;
		Trips_DB.Section[j].Peak.ChargeRelay2_FailtoClose := FALSE;
		Trips_DB.Section[j].Peak.ChargeRelay2_FailtoOpen := FALSE;
		//Sust
		Trips_DB.Section[j].Sust.DumpRelay1_FailtoClose := FALSE;
		Trips_DB.Section[j].Sust.DumpRelay1_FailtoOpen := FALSE;
		Trips_DB.Section[j].Sust.DumpRelay2_FailtoClose := FALSE;
		Trips_DB.Section[j].Sust.DumpRelay2_FailtoOpen := FALSE;
		Trips_DB.Section[j].Sust.ChargeRelay1_FailtoClose := FALSE;
		Trips_DB.Section[j].Sust.ChargeRelay1_FailtoOpen := FALSE;
		Trips_DB.Section[j].Sust.ChargeRelay2_FailtoClose := FALSE;
		Trips_DB.Section[j].Sust.ChargeRelay2_FailtoOpen := FALSE;
	
	END_FOR;
	
	//FORM
	Trips_DB.Section[4].Form.ChargeRelay1_FailtoOpen := FALSE;
	Trips_DB.Section[4].Form.ChargeRelay1_FailtoClose := FALSE;
	Trips_DB.Section[4].Form.ChargeRelay1_Failed:= FALSE;
	Trips_DB.Section[4].Form.ChargeRelay2_FailtoOpen := FALSE;
	Trips_DB.Section[4].Form.ChargeRelay2_FailtoClose := FALSE;
	Trips_DB.Section[4].Form.ChargeRelay2_Failed:= FALSE;
	
	Trips_DB.Section[4].Form.DumpRelay1_FailtoOpen := FALSE;
	Trips_DB.Section[4].Form.DumpRelay1_FailtoClose := FALSE;
	Trips_DB.Section[4].Form.DumpRelay1_Failed := FALSE;
	Trips_DB.Section[4].Form.DumpRelay2_FailtoOpen := FALSE;
	Trips_DB.Section[4].Form.DumpRelay2_FailtoClose := FALSE;
	Trips_DB.Section[4].Form.DumpRelay2_Failed := FALSE;
	
	Trips_DB.Section[4].Form.PreFormChrgRlyFailed := FALSE;
	Trips_DB.Section[4].Form.FormTrigChrgRlyFailed := FALSE;
	Trips_DB.Section[4].Form.PreFormTrigChrgRlyFailed := FALSE;
	Trips_DB.Section[4].Form.PreFormDumpRlyFailed := FALSE;
	Trips_DB.Section[4].Form.FormTrigDumpRly1Failed := FALSE;
	Trips_DB.Section[4].Form.PreFormTrigDumpRly1Failed := FALSE;
	
	Trips_DB.Section[4].SystemTripped := FALSE;
	
	evtLogger.ClearAllAlarms(0, FALSE);
	//evtLogger.ClearLoggedEvents(1);
END_IF;


IF i > 8 THEN 
	i := 1;
END_IF;

IF j > 3 THEN 
	j := 1;
END_IF;

IF k > 4 THEN 
	k := 1;
END_IF;

END_PROGRAM

// ---- POUs/Alarms.TcPOU
PROGRAM Alarms
VAR
	bWarning : BOOL;
	bConfirm : BOOL;
	alarms : ARRAY[0..80] OF Alarms_FB;
	
END_VAR

// Alarm Word 1 - MCP Alarms
//MCP Alarms

Alarms_DB.MCP.AlarmWord.0 := Trips_DB.MasterStopPBPressed;
Alarms_DB.MCP.AlarmWord.1 := Trips_DB.CaseEStopCircuitBroken;
Alarms_DB.MCP.AlarmWord.2 := Trips_DB.ManualModeSelected;
Alarms_DB.MCP.AlarmWord.3 := Trips_DB.MCPLossDCpower;
Alarms_DB.MCP.AlarmWord.4 := MCP_IO.Charger[1].SummaryFaulted;
Alarms_DB.MCP.AlarmWord.5 := MCP_IO.Charger[2].SummaryFaulted;
Alarms_DB.MCP.AlarmWord.6 := MCP_IO.Charger[3].SummaryFaulted;
Alarms_DB.MCP.AlarmWord.7 := MCP_IO.Charger[4].SummaryFaulted;
Alarms_DB.MCP.AlarmWord.8 := MCP_IO.Charger[5].SummaryFaulted;
Alarms_DB.MCP.AlarmWord.9 := MCP_IO.Charger[6].SummaryFaulted;
Alarms_DB.MCP.AlarmWord.10 := MCP_IO.Charger[7].SummaryFaulted;
Alarms_DB.MCP.AlarmWord.11 := MCP_IO.Charger[8].SummaryFaulted;


//Alarm Word 1 msg
//IE: alarms[299](evtEntry:= Tc_Events.AlarmWord11.b4, bEvt:= gvl.test, bConfirm:= bConfirm);
alarms[0](evtEntry:= Tc_Events.AlarmWord1.b0, bEvt:= Alarms_DB.MCP.AlarmWord.0, bConfirm:= bConfirm);
alarms[1](evtEntry:= Tc_Events.AlarmWord1.b1, bEvt:= Alarms_DB.MCP.AlarmWord.1, bConfirm:= bConfirm);
alarms[2](evtEntry:= Tc_Events.AlarmWord1.b2, bEvt:= Alarms_DB.MCP.AlarmWord.2, bConfirm:= bConfirm);
alarms[3](evtEntry:= Tc_Events.AlarmWord1.b3, bEvt:= Alarms_DB.MCP.AlarmWord.3, bConfirm:= bConfirm);
alarms[4](evtEntry:= Tc_Events.AlarmWord1.b4, bEvt:= Alarms_DB.MCP.AlarmWord.4, bConfirm:= bConfirm);
alarms[5](evtEntry:= Tc_Events.AlarmWord1.b5, bEvt:= Alarms_DB.MCP.AlarmWord.5, bConfirm:= bConfirm);
alarms[6](evtEntry:= Tc_Events.AlarmWord1.b6, bEvt:= Alarms_DB.MCP.AlarmWord.6, bConfirm:= bConfirm);
alarms[7](evtEntry:= Tc_Events.AlarmWord1.b7, bEvt:= Alarms_DB.MCP.AlarmWord.7, bConfirm:= bConfirm);
alarms[8](evtEntry:= Tc_Events.AlarmWord1.b8, bEvt:= Alarms_DB.MCP.AlarmWord.8, bConfirm:= bConfirm);
alarms[9](evtEntry:= Tc_Events.AlarmWord1.b9, bEvt:= Alarms_DB.MCP.AlarmWord.9, bConfirm:= bConfirm);
alarms[0](evtEntry:= Tc_Events.AlarmWord1.b10, bEvt:= Alarms_DB.MCP.AlarmWord.10, bConfirm:= bConfirm);
alarms[11](evtEntry:= Tc_Events.AlarmWord1.b11, bEvt:= Alarms_DB.MCP.AlarmWord.11, bConfirm:= bConfirm);
//alarms[12] - spare
//alarms[13] - spare
//alarms[14] - spare
//alarms[15] - spare

// Alarm Word 2 - Section 1 Alarms
Alarms_DB.Section1.AlarmWord.0 := Trips_DB.Section[1].SystemTripped;
Alarms_DB.Section1.AlarmWord.1 := Trips_DB.Section[1].LossPneumaticPressure;
Alarms_DB.Section1.AlarmWord.2 := Trips_DB.Section[1].Peak.ChargeRelay1_Failed;
Alarms_DB.Section1.AlarmWord.3 := Trips_DB.Section[1].Peak.ChargeRelay2_Failed;
Alarms_DB.Section1.AlarmWord.4 := Trips_DB.Section[1].Peak.DumpRelay1_Failed;
Alarms_DB.Section1.AlarmWord.5 := Trips_DB.Section[1].Peak.DumpRelay2_Failed;
Alarms_DB.Section1.AlarmWord.6 := Trips_DB.Section[1].Sust.ChargeRelay1_Failed;
Alarms_DB.Section1.AlarmWord.7 := Trips_DB.Section[1].Sust.ChargeRelay2_Failed;
Alarms_DB.Section1.AlarmWord.8 := Trips_DB.Section[1].Sust.DumpRelay1_Failed;
Alarms_DB.Section1.AlarmWord.9 := Trips_DB.Section[1].Sust.DumpRelay2_Failed;
Alarms_DB.Section1.AlarmWord.10 := Trips_DB.Section[1].LossDCPower;


// Alarm Word 2 - Msg
alarms[16](evtEntry:= Tc_Events.AlarmWord2.b0, bEvt:= Alarms_DB.Section1.AlarmWord.0, bConfirm:= bConfirm);
alarms[17](evtEntry:= Tc_Events.AlarmWord2.b1, bEvt:= Alarms_DB.Section1.AlarmWord.1, bConfirm:= bConfirm);
alarms[18](evtEntry:= Tc_Events.AlarmWord2.b2, bEvt:= Alarms_DB.Section1.AlarmWord.2, bConfirm:= bConfirm);
alarms[19](evtEntry:= Tc_Events.AlarmWord2.b3, bEvt:= Alarms_DB.Section1.AlarmWord.3, bConfirm:= bConfirm);
alarms[20](evtEntry:= Tc_Events.AlarmWord2.b4, bEvt:= Alarms_DB.Section1.AlarmWord.4, bConfirm:= bConfirm);
alarms[21](evtEntry:= Tc_Events.AlarmWord2.b5, bEvt:= Alarms_DB.Section1.AlarmWord.5, bConfirm:= bConfirm);
alarms[22](evtEntry:= Tc_Events.AlarmWord2.b6, bEvt:= Alarms_DB.Section1.AlarmWord.6, bConfirm:= bConfirm);
alarms[23](evtEntry:= Tc_Events.AlarmWord2.b7, bEvt:= Alarms_DB.Section1.AlarmWord.7, bConfirm:= bConfirm);
alarms[24](evtEntry:= Tc_Events.AlarmWord2.b8, bEvt:= Alarms_DB.Section1.AlarmWord.8, bConfirm:= bConfirm);
alarms[25](evtEntry:= Tc_Events.AlarmWord2.b9, bEvt:= Alarms_DB.Section1.AlarmWord.9, bConfirm:= bConfirm);
alarms[26](evtEntry:= Tc_Events.AlarmWord2.b10, bEvt:= Alarms_DB.Section1.AlarmWord.10, bConfirm:= bConfirm);
//alarms[27] - spare
//alarms[28] - spare
//alarms[29] - spare
//alarms[30] - spare
//alarms[31] - spare


// Alarm Word 3 - Section 2 Alarms
Alarms_DB.Section2.AlarmWord.0 := Trips_DB.Section[2].SystemTripped;
Alarms_DB.Section2.AlarmWord.1 := Trips_DB.Section[2].LossPneumaticPressure;
Alarms_DB.Section2.AlarmWord.2 := Trips_DB.Section[2].Peak.ChargeRelay1_Failed;
Alarms_DB.Section2.AlarmWord.3 := Trips_DB.Section[2].Peak.ChargeRelay2_Failed;
Alarms_DB.Section2.AlarmWord.4 := Trips_DB.Section[2].Peak.DumpRelay1_Failed;
Alarms_DB.Section2.AlarmWord.5 := Trips_DB.Section[2].Peak.DumpRelay2_Failed;
Alarms_DB.Section2.AlarmWord.6 := Trips_DB.Section[2].Sust.ChargeRelay1_Failed;
Alarms_DB.Section2.AlarmWord.7 := Trips_DB.Section[2].Sust.ChargeRelay2_Failed;
Alarms_DB.Section2.AlarmWord.8 := Trips_DB.Section[2].Sust.DumpRelay1_Failed;
Alarms_DB.Section2.AlarmWord.9 := Trips_DB.Section[2].Sust.DumpRelay2_Failed;
Alarms_DB.Section2.AlarmWord.10 := Trips_DB.Section[2].LossDCPower;


// Alarm Word 3 - Msg
alarms[32](evtEntry:= Tc_Events.AlarmWord3.b0, bEvt:= Alarms_DB.Section2.AlarmWord.0, bConfirm:= bConfirm);
alarms[33](evtEntry:= Tc_Events.AlarmWord3.b1, bEvt:= Alarms_DB.Section2.AlarmWord.1, bConfirm:= bConfirm);
alarms[34](evtEntry:= Tc_Events.AlarmWord3.b2, bEvt:= Alarms_DB.Section2.AlarmWord.2, bConfirm:= bConfirm);
alarms[35](evtEntry:= Tc_Events.AlarmWord3.b3, bEvt:= Alarms_DB.Section2.AlarmWord.3, bConfirm:= bConfirm);
alarms[36](evtEntry:= Tc_Events.AlarmWord3.b4, bEvt:= Alarms_DB.Section2.AlarmWord.4, bConfirm:= bConfirm);
alarms[37](evtEntry:= Tc_Events.AlarmWord3.b5, bEvt:= Alarms_DB.Section2.AlarmWord.5, bConfirm:= bConfirm);
alarms[38](evtEntry:= Tc_Events.AlarmWord3.b6, bEvt:= Alarms_DB.Section2.AlarmWord.6, bConfirm:= bConfirm);
alarms[39](evtEntry:= Tc_Events.AlarmWord3.b7, bEvt:= Alarms_DB.Section2.AlarmWord.7, bConfirm:= bConfirm);
alarms[40](evtEntry:= Tc_Events.AlarmWord3.b8, bEvt:= Alarms_DB.Section2.AlarmWord.8, bConfirm:= bConfirm);
alarms[41](evtEntry:= Tc_Events.AlarmWord3.b9, bEvt:= Alarms_DB.Section2.AlarmWord.9, bConfirm:= bConfirm);
alarms[42](evtEntry:= Tc_Events.AlarmWord3.b10, bEvt:= Alarms_DB.Section2.AlarmWord.10, bConfirm:= bConfirm);
//alarms[43] - spare
//alarms[44] - spare
//alarms[45] - spare
//alarms[46] - spare
//alarms[47] - spare

// Alarm Word 4 - Section 3 Alarms
Alarms_DB.Section3.AlarmWord.0 := Trips_DB.Section[3].SystemTripped;
Alarms_DB.Section3.AlarmWord.1 := Trips_DB.Section[3].LossPneumaticPressure;
Alarms_DB.Section3.AlarmWord.2 := Trips_DB.Section[3].Peak.ChargeRelay1_Failed;
Alarms_DB.Section3.AlarmWord.3 := Trips_DB.Section[3].Peak.ChargeRelay2_Failed;
Alarms_DB.Section3.AlarmWord.4 := Trips_DB.Section[3].Peak.DumpRelay1_Failed;
Alarms_DB.Section3.AlarmWord.5 := Trips_DB.Section[3].Peak.DumpRelay2_Failed;
Alarms_DB.Section3.AlarmWord.6 := Trips_DB.Section[3].Sust.ChargeRelay1_Failed;
Alarms_DB.Section3.AlarmWord.7 := Trips_DB.Section[3].Sust.ChargeRelay2_Failed;
Alarms_DB.Section3.AlarmWord.8 := Trips_DB.Section[3].Sust.DumpRelay1_Failed;
Alarms_DB.Section3.AlarmWord.9 := Trips_DB.Section[3].Sust.DumpRelay2_Failed;
Alarms_DB.Section3.AlarmWord.10 := Trips_DB.Section[3].LossDCPower;


// Alarm Word 4 - Msg
alarms[48](evtEntry:= Tc_Events.AlarmWord4.b0, bEvt:= Alarms_DB.Section3.AlarmWord.0, bConfirm:= bConfirm);
alarms[49](evtEntry:= Tc_Events.AlarmWord4.b1, bEvt:= Alarms_DB.Section3.AlarmWord.1, bConfirm:= bConfirm);
alarms[50](evtEntry:= Tc_Events.AlarmWord4.b2, bEvt:= Alarms_DB.Section3.AlarmWord.2, bConfirm:= bConfirm);
alarms[51](evtEntry:= Tc_Events.AlarmWord4.b3, bEvt:= Alarms_DB.Section3.AlarmWord.3, bConfirm:= bConfirm);
alarms[52](evtEntry:= Tc_Events.AlarmWord4.b4, bEvt:= Alarms_DB.Section3.AlarmWord.4, bConfirm:= bConfirm);
alarms[53](evtEntry:= Tc_Events.AlarmWord4.b5, bEvt:= Alarms_DB.Section3.AlarmWord.5, bConfirm:= bConfirm);
alarms[54](evtEntry:= Tc_Events.AlarmWord4.b6, bEvt:= Alarms_DB.Section3.AlarmWord.6, bConfirm:= bConfirm);
alarms[55](evtEntry:= Tc_Events.AlarmWord4.b7, bEvt:= Alarms_DB.Section3.AlarmWord.7, bConfirm:= bConfirm);
alarms[56](evtEntry:= Tc_Events.AlarmWord4.b8, bEvt:= Alarms_DB.Section3.AlarmWord.8, bConfirm:= bConfirm);
alarms[57](evtEntry:= Tc_Events.AlarmWord4.b9, bEvt:= Alarms_DB.Section3.AlarmWord.9, bConfirm:= bConfirm);
alarms[58](evtEntry:= Tc_Events.AlarmWord4.b10, bEvt:= Alarms_DB.Section3.AlarmWord.10, bConfirm:= bConfirm);
//alarms[59] - spare
//alarms[60] - spare
//alarms[61] - spare
//alarms[62] - spare
//alarms[63] - spare

// Alarm Word 5 - Section 4 Alarms
Alarms_DB.Section4.AlarmWord.0 := Trips_DB.Section[4].SystemTripped;
Alarms_DB.Section4.AlarmWord.1 := Trips_DB.Section[4].LossPneumaticPressure;
Alarms_DB.Section4.AlarmWord.2 := Trips_DB.Section[4].Form.ChargeRelay1_Failed;
Alarms_DB.Section4.AlarmWord.3 := Trips_DB.Section[4].Form.ChargeRelay2_Failed;
Alarms_DB.Section4.AlarmWord.4 := Trips_DB.Section[4].Form.DumpRelay1_Failed;
Alarms_DB.Section4.AlarmWord.5 := Trips_DB.Section[4].Form.DumpRelay2_Failed;
Alarms_DB.Section4.AlarmWord.6 := Trips_DB.Section[4].Form.PreFormChrgRlyFailed;
Alarms_DB.Section4.AlarmWord.7 := Trips_DB.Section[4].Form.FormTrigChrgRlyFailed;
Alarms_DB.Section4.AlarmWord.8 := Trips_DB.Section[4].Form.PreFormTrigChrgRlyFailed;
Alarms_DB.Section4.AlarmWord.9 := Trips_DB.Section[4].Form.PreFormDumpRlyFailed;
Alarms_DB.Section4.AlarmWord.10 := Trips_DB.Section[4].Form.FormTrigDumpRly1Failed;
Alarms_DB.Section4.AlarmWord.11 := Trips_DB.Section[4].Form.PreFormTrigDumpRly1Failed;
Alarms_DB.Section4.AlarmWord.12 := Trips_DB.Section[4].LossDCPower;

// Alarm Word 5 - Msg
alarms[64](evtEntry:= Tc_Events.AlarmWord5.b0, bEvt:= Alarms_DB.Section4.AlarmWord.0, bConfirm:= bConfirm);
alarms[65](evtEntry:= Tc_Events.AlarmWord5.b1, bEvt:= Alarms_DB.Section4.AlarmWord.1, bConfirm:= bConfirm);
alarms[66](evtEntry:= Tc_Events.AlarmWord5.b2, bEvt:= Alarms_DB.Section4.AlarmWord.2, bConfirm:= bConfirm);
alarms[67](evtEntry:= Tc_Events.AlarmWord5.b3, bEvt:= Alarms_DB.Section4.AlarmWord.3, bConfirm:= bConfirm);
alarms[68](evtEntry:= Tc_Events.AlarmWord5.b4, bEvt:= Alarms_DB.Section4.AlarmWord.4, bConfirm:= bConfirm);
alarms[69](evtEntry:= Tc_Events.AlarmWord5.b5, bEvt:= Alarms_DB.Section4.AlarmWord.5, bConfirm:= bConfirm);
alarms[70](evtEntry:= Tc_Events.AlarmWord5.b6, bEvt:= Alarms_DB.Section4.AlarmWord.6, bConfirm:= bConfirm);
alarms[71](evtEntry:= Tc_Events.AlarmWord5.b7, bEvt:= Alarms_DB.Section4.AlarmWord.7, bConfirm:= bConfirm);
alarms[72](evtEntry:= Tc_Events.AlarmWord5.b8, bEvt:= Alarms_DB.Section4.AlarmWord.8, bConfirm:= bConfirm);
alarms[73](evtEntry:= Tc_Events.AlarmWord5.b9, bEvt:= Alarms_DB.Section4.AlarmWord.9, bConfirm:= bConfirm);
alarms[74](evtEntry:= Tc_Events.AlarmWord5.b10, bEvt:= Alarms_DB.Section4.AlarmWord.10, bConfirm:= bConfirm);
alarms[75](evtEntry:= Tc_Events.AlarmWord5.b10, bEvt:= Alarms_DB.Section4.AlarmWord.11, bConfirm:= bConfirm);
alarms[76](evtEntry:= Tc_Events.AlarmWord5.b10, bEvt:= Alarms_DB.Section4.AlarmWord.12, bConfirm:= bConfirm);
//alarms[77] - spare
//alarms[78] - spare
//alarms[79] - spare


//Alarm Word 11
(* uncomment this when instrument is ready
Alarms_DB.AlarmWord_11.AlarmWord.0 := Devices.Coil1.AC_Interlock_RlyOpen;
Alarms_DB.AlarmWord_11.AlarmWord.1 := Devices.Coil2.AC_Interlock_RlyOpen;
Alarms_DB.AlarmWord_11.AlarmWord.2 := Devices.Coil3.AC_Interlock_RlyOpen;
Alarms_DB.AlarmWord_11.AlarmWord.3 := Devices.Coil4.AC_Interlock_RlyOpen;
Alarms_DB.AlarmWord_11.AlarmWord.4 := Devices.Coil5.AC_Interlock_RlyOpen;
Alarms_DB.AlarmWord_11.AlarmWord.5 := Devices.Coil6.AC_Interlock_RlyOpen;
Alarms_DB.AlarmWord_11.AlarmWord.6 := Devices.Coil7.AC_Interlock_RlyOpen;
Alarms_DB.AlarmWord_11.AlarmWord.7 := Devices.Coil8.AC_Interlock_RlyOpen;
Alarms_DB.AlarmWord_11.AlarmWord.8 := Devices.Coil9.AC_Interlock_RlyOpen;
Alarms_DB.AlarmWord_11.AlarmWord.9 := Devices.Coil10.AC_Interlock_RlyOpen;
Alarms_DB.AlarmWord_11.AlarmWord.10 := NOT Permissives.AllInterlock_Closed;
*)
//Alarm Word 11 - msg
(*alarms[160](evtEntry:= Tc_Events.AlarmWord11.b0, bEvt:= Alarms_DB.AlarmWord_11.AlarmWord.0, bConfirm:= bConfirm);
alarms[161](evtEntry:= Tc_Events.AlarmWord11.b1, bEvt:= Alarms_DB.AlarmWord_11.AlarmWord.1, bConfirm:= bConfirm);
alarms[162](evtEntry:= Tc_Events.AlarmWord11.b2, bEvt:= Alarms_DB.AlarmWord_11.AlarmWord.2, bConfirm:= bConfirm);
alarms[163](evtEntry:= Tc_Events.AlarmWord11.b3, bEvt:= Alarms_DB.AlarmWord_11.AlarmWord.3, bConfirm:= bConfirm);
alarms[164](evtEntry:= Tc_Events.AlarmWord11.b4, bEvt:= Alarms_DB.AlarmWord_11.AlarmWord.4, bConfirm:= bConfirm);
alarms[165](evtEntry:= Tc_Events.AlarmWord11.b5, bEvt:= Alarms_DB.AlarmWord_11.AlarmWord.5, bConfirm:= bConfirm);
alarms[166](evtEntry:= Tc_Events.AlarmWord11.b6, bEvt:= Alarms_DB.AlarmWord_11.AlarmWord.6, bConfirm:= bConfirm);
alarms[167](evtEntry:= Tc_Events.AlarmWord11.b7, bEvt:= Alarms_DB.AlarmWord_11.AlarmWord.7, bConfirm:= bConfirm);
alarms[168](evtEntry:= Tc_Events.AlarmWord11.b8, bEvt:= Alarms_DB.AlarmWord_11.AlarmWord.8, bConfirm:= bConfirm);
alarms[169](evtEntry:= Tc_Events.AlarmWord11.b9, bEvt:= Alarms_DB.AlarmWord_11.AlarmWord.9, bConfirm:= bConfirm);
alarms[170](evtEntry:= Tc_Events.AlarmWord11.b10, bEvt:= Alarms_DB.AlarmWord_11.AlarmWord.10, bConfirm:= bConfirm);

//Alarm Word 12




//Alarm Word 22
//uncomment this when instrument is ready - commented out for testing only
Alarms_DB.AlarmWord_22.AlarmWord.0 := MCP_IO.MasterStopPB_Pressed; //NC
(*//Alarms_DB1.AlarmWord_22.AlarmWord.1 := Devices.Coil[1].Local_EstopPB_Pressed; //NC
Alarms_DB1.AlarmWord_22.AlarmWord.2 := Devices.Coil2.Local_EstopPB_Pressed; //NC
Alarms_DB1.AlarmWord_22.AlarmWord.3 := Devices.Coil3.Local_EstopPB_Pressed; //NC
Alarms_DB1.AlarmWord_22.AlarmWord.4 := Devices.Coil4.Local_EstopPB_Pressed; //NC
Alarms_DB1.AlarmWord_22.AlarmWord.5 := Devices.Coil5.Local_EstopPB_Pressed; //NC
Alarms_DB1.AlarmWord_22.AlarmWord.6 := Devices.Coil6.Local_EstopPB_Pressed; //NC
Alarms_DB1.AlarmWord_22.AlarmWord.7 := Devices.Coil7.Local_EstopPB_Pressed; //NC
Alarms_DB1.AlarmWord_22.AlarmWord.8 := Devices.Coil8.Local_EstopPB_Pressed; //NC
Alarms_DB1.AlarmWord_22.AlarmWord.9 := Devices.Coil9.Local_EstopPB_Pressed; //NC
Alarms_DB1.AlarmWord_22.AlarmWord.10 := Devices.Coil10.Local_EstopPB_Pressed; //NC
//Alarms_DB1.AlarmWord_22.AlarmWord.11 := NOT Input.R1_01_02; //0 = Manual Mode , 1 = Auto mode
//Alarms_DB1.AlarmWord_22.AlarmWord.12 := NOT Input.R1_01_01; //0 = circuit broken , 1 = circuit ok
//Alarms_DB1.AlarmWord_22.AlarmWord.13 := Spare
//Alarms_DB1.AlarmWord_22.AlarmWord.14 := Spare
//Alarms_DB1.AlarmWord_22.AlarmWord.15 := Spare
*)

//Alarm Word 22 msg
alarms[336](evtEntry:= Tc_Events.AlarmWord22.b0, bEvt:= Alarms_DB.AlarmWord_22.AlarmWord.0, bConfirm:= bConfirm);
alarms[337](evtEntry:= Tc_Events.AlarmWord22.b1, bEvt:= Alarms_DB.AlarmWord_22.AlarmWord.1, bConfirm:= bConfirm);
alarms[338](evtEntry:= Tc_Events.AlarmWord22.b2, bEvt:= Alarms_DB.AlarmWord_22.AlarmWord.2, bConfirm:= bConfirm);
alarms[339](evtEntry:= Tc_Events.AlarmWord22.b3, bEvt:= Alarms_DB.AlarmWord_22.AlarmWord.3, bConfirm:= bConfirm);
alarms[340](evtEntry:= Tc_Events.AlarmWord22.b4, bEvt:= Alarms_DB.AlarmWord_22.AlarmWord.4, bConfirm:= bConfirm);
alarms[341](evtEntry:= Tc_Events.AlarmWord22.b5, bEvt:= Alarms_DB.AlarmWord_22.AlarmWord.5, bConfirm:= bConfirm);
alarms[342](evtEntry:= Tc_Events.AlarmWord22.b6, bEvt:= Alarms_DB.AlarmWord_22.AlarmWord.6, bConfirm:= bConfirm);
alarms[343](evtEntry:= Tc_Events.AlarmWord22.b7, bEvt:= Alarms_DB.AlarmWord_22.AlarmWord.7, bConfirm:= bConfirm);
alarms[344](evtEntry:= Tc_Events.AlarmWord22.b8, bEvt:= Alarms_DB.AlarmWord_22.AlarmWord.8, bConfirm:= bConfirm);
alarms[345](evtEntry:= Tc_Events.AlarmWord22.b9, bEvt:= Alarms_DB.AlarmWord_22.AlarmWord.9, bConfirm:= bConfirm);
alarms[346](evtEntry:= Tc_Events.AlarmWord22.b10, bEvt:= Alarms_DB.AlarmWord_22.AlarmWord.10, bConfirm:= bConfirm);
alarms[347](evtEntry:= Tc_Events.AlarmWord22.b11, bEvt:= Alarms_DB.AlarmWord_22.AlarmWord.11, bConfirm:= bConfirm);
alarms[348](evtEntry:= Tc_Events.AlarmWord22.b12, bEvt:= Alarms_DB.AlarmWord_22.AlarmWord.12, bConfirm:= bConfirm);

//Alarm Word 23
(* uncomment when instrument is ready
Alarms_DB.AlarmWord_23.AlarmWord.0 := Trips_DB.Coil[1].ChargeRelay_FailtoClose; 
Alarms_DB.AlarmWord_23.AlarmWord.1 := Trips_DB.Coil[1].ChargeRelay_FailtoOpen;
Alarms_DB.AlarmWord_23.AlarmWord.2 := Trips_DB.Coil[2].ChargeRelay_FailtoClose;
Alarms_DB.AlarmWord_23.AlarmWord.3 := Trips_DB.Coil[2].ChargeRelay_FailtoOpen;
Alarms_DB.AlarmWord_23.AlarmWord.4 := Trips_DB.Coil[3].ChargeRelay_FailtoClose;
Alarms_DB.AlarmWord_23.AlarmWord.5 := Trips_DB.Coil[3].ChargeRelay_FailtoOpen;
Alarms_DB.AlarmWord_23.AlarmWord.6 := Trips_DB.Coil[4].ChargeRelay_FailtoClose;
Alarms_DB.AlarmWord_23.AlarmWord.7 := Trips_DB.Coil[4].ChargeRelay_FailtoOpen;
Alarms_DB.AlarmWord_23.AlarmWord.8 := Trips_DB.Coil[5].ChargeRelay_FailtoClose;
Alarms_DB.AlarmWord_23.AlarmWord.9 := Trips_DB.Coil[5].ChargeRelay_FailtoOpen;
Alarms_DB.AlarmWord_23.AlarmWord.10 := Trips_DB.Coil[6].ChargeRelay_FailtoClose;
Alarms_DB.AlarmWord_23.AlarmWord.11 := Trips_DB.Coil[6].ChargeRelay_FailtoOpen;
Alarms_DB.AlarmWord_23.AlarmWord.12 := Trips_DB.Coil[7].ChargeRelay_FailtoClose;
Alarms_DB.AlarmWord_23.AlarmWord.13 := Trips_DB.Coil[7].ChargeRelay_FailtoOpen;
Alarms_DB.AlarmWord_23.AlarmWord.14 := Trips_DB.Coil[8].ChargeRelay_FailtoClose;
Alarms_DB.AlarmWord_23.AlarmWord.15 := Trips_DB.Coil[9].ChargeRelay_FailtoOpen;
*)
//Alarm Word 23 msg
alarms[352](evtEntry:= Tc_Events.AlarmWord23.b0, bEvt:= Alarms_DB.AlarmWord_23.AlarmWord.0, bConfirm:= bConfirm);
alarms[353](evtEntry:= Tc_Events.AlarmWord23.b1, bEvt:= Alarms_DB.AlarmWord_23.AlarmWord.1, bConfirm:= bConfirm);
alarms[354](evtEntry:= Tc_Events.AlarmWord23.b2, bEvt:= Alarms_DB.AlarmWord_23.AlarmWord.2, bConfirm:= bConfirm);
alarms[355](evtEntry:= Tc_Events.AlarmWord23.b3, bEvt:= Alarms_DB.AlarmWord_23.AlarmWord.3, bConfirm:= bConfirm);
alarms[356](evtEntry:= Tc_Events.AlarmWord23.b4, bEvt:= Alarms_DB.AlarmWord_23.AlarmWord.4, bConfirm:= bConfirm);
alarms[357](evtEntry:= Tc_Events.AlarmWord23.b5, bEvt:= Alarms_DB.AlarmWord_23.AlarmWord.5, bConfirm:= bConfirm);
alarms[358](evtEntry:= Tc_Events.AlarmWord23.b6, bEvt:= Alarms_DB.AlarmWord_23.AlarmWord.6, bConfirm:= bConfirm);
alarms[359](evtEntry:= Tc_Events.AlarmWord23.b7, bEvt:= Alarms_DB.AlarmWord_23.AlarmWord.7, bConfirm:= bConfirm);
alarms[360](evtEntry:= Tc_Events.AlarmWord23.b8, bEvt:= Alarms_DB.AlarmWord_23.AlarmWord.8, bConfirm:= bConfirm);
alarms[361](evtEntry:= Tc_Events.AlarmWord23.b9, bEvt:= Alarms_DB.AlarmWord_23.AlarmWord.9, bConfirm:= bConfirm);
alarms[362](evtEntry:= Tc_Events.AlarmWord23.b10, bEvt:= Alarms_DB.AlarmWord_23.AlarmWord.10, bConfirm:= bConfirm);
alarms[363](evtEntry:= Tc_Events.AlarmWord23.b11, bEvt:= Alarms_DB.AlarmWord_23.AlarmWord.11, bConfirm:= bConfirm);
alarms[364](evtEntry:= Tc_Events.AlarmWord23.b12, bEvt:= Alarms_DB.AlarmWord_23.AlarmWord.12, bConfirm:= bConfirm);
alarms[365](evtEntry:= Tc_Events.AlarmWord23.b13, bEvt:= Alarms_DB.AlarmWord_23.AlarmWord.13, bConfirm:= bConfirm);
alarms[366](evtEntry:= Tc_Events.AlarmWord23.b14, bEvt:= Alarms_DB.AlarmWord_23.AlarmWord.14, bConfirm:= bConfirm);
alarms[367](evtEntry:= Tc_Events.AlarmWord23.b15, bEvt:= Alarms_DB.AlarmWord_23.AlarmWord.15, bConfirm:= bConfirm);

